Private helper method that removes the oldest element from the list based on the
fill direction. This method is called by Push() when the buffer is full to make
space for a new element.

### Operation
- fillFromLeft = TRUE: Oldest at end (high index), uses PopRight
- fillFromLeft = FALSE: Oldest at front (index 0), uses PopLeft

The removed element is discarded as we only care about making space.

### Return Value
- **TRUE**: Oldest element was successfully removed
- **FALSE**: Remove operation failed

### Side Effects
- Removes one element from the list
- May shift remaining elements (fillFromLeft = FALSE)
- Decrements element count by 1
- Increases available capacity by 1
*)
removeOldest := FALSE;
IF _reversed THEN
	// Fill from left: oldest element is at the end (highest index)
	removeOldest := anyBuffer.PopRight(dummyElement, TRUE);
ELSE
	// Fill from right: oldest element is at the front (index 0)
	removeOldest := anyBuffer.PopLeft(dummyElement, TRUE);
END_IF
END_METHOD

END_FUNCTION_BLOCK

// ---- Utilities/AnyBuffer/TypedBuffers/RingBuffer.TcPOU
// Provides a circular buffer (ring buffer) interface with automatic overwrite capability
FUNCTION_BLOCK RingBuffer IMPLEMENTS I_AnyBufferStrategy
VAR
	anyBuffer	  : I_AnyBuffer;
	isInitialized : BOOL := FALSE;
	_overwrite	  : BOOL := TRUE; // TRUE: overwrites oldest when full
END_VAR

(*
## Detailed Description

RingBuffer is an adapter that wraps an AnyBuffer instance to provide circular buffer
(also called ring buffer) semantics with automatic overwrite capability. When the buffer
is full and a new element is added, the oldest element is automatically removed to make
space, creating a continuous circular data flow.

### Alternative Names
This data structure is commonly known as:
- **Ring Buffer**: Emphasizes the circular/wrap-around nature
- **Circular Buffer**: Describes the logical circular structure
- **Cyclic Buffer**: Another term for the same concept

### Design Pattern
This implements the **Adapter Pattern**, which:
- Wraps the AnyBuffer interface with domain-specific circular buffer semantics
- Delegates all operations to the underlying AnyBuffer instance
- Provides automatic overwrite behavior when buffer reaches capacity
- Useful for streaming data, logging, and producer-consumer patterns

### Ring Buffer Semantics
- **Push(element)**: Adds element using circular indexing (FIFO enqueue)
  - When not full: Uses WriteAtIndex for direct write at tail position
  - When full: Overwrites oldest element using WriteAtIndex (no shifting!)
- **Pop(element)**: Removes oldest element using PeekAtIndex and circular head pointer (no shifting!)
- **Automatic overwrite**: When enabled and buffer is full, oldest data is overwritten in place
- **Circular indexing**: Uses head/tail pointers to track logical queue positions
- **Direct memory access**: Uses WriteAtIndex for O(1) writes without counter overhead
- Elements maintain FIFO order (first in, first out)

### Operation Mapping
```
Push() when not full  -> anyBuffer.WriteAtIndex(tail, ...)  // Direct write (O(1), no counter overhead)
Push() when full      -> anyBuffer.WriteAtIndex(tail, ...)  // Overwrite oldest (O(1), no shift!)
Pop()                 -> anyBuffer.PeekAtIndex(head, ...)   // Read oldest (O(1), no shift!)
Clear()               -> anyBuffer.Clear()                  // Clear all + reset indices
isEmpty               -> (elementCount = 0)                 // Check element count
isFull                -> (elementCount >= capacity)         // Check element count
```

### Usage Example
```iecst
VAR
    rawBuffer : ARRAY[0..2] OF DINT;  // Small buffer for demonstration
    buffer : AnyBuffer(pBuffer := rawBuffer,
                       bufferBoundLower := 0,
                       bufferBoundUpper := 2,
                       isBufferPersistent := FALSE);
    ring : RingBuffer(anyBuffer := buffer, overwrite := TRUE);
    value : DINT;
END_VAR

// Fill buffer
value := 100; ring.Push(value);  // Buffer: [100]
value := 200; ring.Push(value);  // Buffer: [100, 200]
value := 300; ring.Push(value);  // Buffer: [100, 200, 300] (full)

// Push to full buffer - oldest (100) is automatically removed
value := 400; ring.Push(value);  // Buffer: [200, 300, 400]
value := 500; ring.Push(value);  // Buffer: [300, 400, 500]

// Pop retrieves in FIFO order
ring.Pop(value);  // value = 300, Buffer: [400, 500]
```

### Circular Buffer Visualization
```
Initial state (capacity 5):
[ ][ ][ ][ ][ ]

After pushing 100, 200, 300:
[100][200][300][ ][ ]

After filling completely (100, 200, 300, 400, 500):
[100][200][300][400][500]  <- Full

After pushing 600 (overwrites 100):
[600][200][300][400][500]
     ^                ^
   oldest          newest

After pushing 700 (overwrites 200):
[600][700][300][400][500]
          ^             ^
       oldest       newest
```

### Advantages
- **No data loss when streaming**: Automatically maintains most recent data
- **Constant memory usage**: Buffer size never grows beyond capacity
- **Highly efficient**: Both Push and Pop are O(1) with circular indexing (no shifting!)
- **Simple interface**: Push/Pop semantics like FifoBuffer
- **Predictable behavior**: Always keeps newest data when overwrite is enabled
- **True circular buffer**: Implements proper ring buffer with head/tail pointers

### Use Cases
- **Logging buffers**: Keep most recent N log messages
- **Sensor data streams**: Store latest readings, discard old data
- **Audio/video buffers**: Maintain continuous data flow
- **Producer-consumer patterns**: Decouple data production and consumption rates
- **History tracking**: Keep fixed-size history of events or states

### Comparison with FifoBuffer
| Feature | FifoBuffer | RingBuffer |
|---------|-----------|------------|
| Behavior when full | Rejects new elements | Overwrites oldest |
| Push operation | Fails if full | Always succeeds |
| Data loss | Never (rejects push) | Yes (by design) |
| Use case | Queue with backpressure | Streaming data |
| Memory | Fixed size | Fixed size |

### Overwrite Behavior
- **overwrite = TRUE**: Push to full buffer removes oldest, adds newest (circular)
- **overwrite = FALSE**: Push to full buffer fails (same as FifoBuffer)

### Limitations
- No random access: Cannot peek at arbitrary indices (use AnyBuffer directly if needed)
- Overwrite is automatic: Cannot prevent data loss when buffer is full (by design)
- No notification: Caller is not informed when overwrite occurs

### Dependencies
- Requires I_AnyBuffer implementation (e.g., AnyBuffer)
- Uses Trace for error logging and verbose diagnostics
- Implements I_AnyBufferStrategy interface

### Performance Considerations
- **Push when not full**: O(1) - uses AppendRight
- **Push when full**: O(1) - uses ReplaceAtIndex with circular indexing (no shifting!)
- **Pop**: O(1) - uses PeekAtIndex with circular indexing (no shifting!)
- **Overall**: True O(1) constant-time operations for all Push and Pop operations
- Ideal for high-performance scenarios with frequent overwrites and streaming data

### Related Patterns
- **FifoBuffer**: FIFO queue without overwrite (rejects when full)
- **LifoBuffer**: Stack (Last-In-First-Out) semantics
- **PriorityBuffer**: Priority queue with ordered insertion
*)

METHOD PRIVATE AdvanceHead
// Advance tail pointer (circular)
anyBuffer.Metadata.headIndex := anyBuffer.Metadata.headIndex + 1;
IF anyBuffer.Metadata.headIndex > anyBuffer.Configuration.bufferBoundUpper THEN
	anyBuffer.Metadata.headIndex := anyBuffer.Configuration.bufferBoundLower;
END_IF
END_METHOD

METHOD PRIVATE AdvanceTail
// Advance tail pointer (circular)
anyBuffer.Metadata.tailIndex := anyBuffer.Metadata.tailIndex + 1;
IF anyBuffer.Metadata.tailIndex > anyBuffer.Configuration.bufferBoundUpper THEN
	anyBuffer.Metadata.tailIndex := anyBuffer.Configuration.bufferBoundLower;
END_IF
END_METHOD

// Removes all elements from the ring buffer and resets to empty state
METHOD Clear : BOOL

(*
## Detailed Description

Clears all elements from the underlying buffer, resetting it to an empty state.
After calling Clear, isEmpty will return TRUE and elementCount will be 0.

This operation delegates directly to the underlying anyBuffer.Clear() method.

### Return Value
- **TRUE**: Ring buffer was successfully cleared
- **FALSE**: Clear operation failed (e.g., anyBuffer is not initialized)

### Side Effects
- All elements are removed from the buffer
- Element count is reset to 0
- Buffer capacity is restored to maximum
- Logs verbose trace message on success
*)
Clear := FALSE;
IF anyBuffer <> 0 THEN
	Clear := anyBuffer.Clear();

	// Reset circular buffer indices
	anyBuffer.Metadata.headIndex	:= anyBuffer.Configuration.bufferBoundLower;
	anyBuffer.Metadata.tailIndex	:= anyBuffer.Configuration.bufferBoundLower;
	anyBuffer.Metadata.elementCount := 0;
END_IF

Trace.Verbose(__POUNAME(), 'executed');
END_METHOD

// Initializes the ring buffer by injecting the underlying buffer dependency
METHOD FB_Init : BOOL
VAR_INPUT
	bInitRetains : BOOL;		 // TRUE: the retain variables are initialized (reset warm / reset cold)
	bInCopyCode	 : BOOL;		 // TRUE: the instance will be copied to the copy code afterward (online change)
	anyBuffer	 : I_AnyBuffer;	 // The underlying buffer implementation to wrap
	overwrite	 : BOOL := TRUE; // TRUE: overwrites oldest element when full (circular behavior)
END_VAR

(*
## Detailed Description

Initializes the RingBuffer by injecting the underlying AnyBuffer dependency. This follows
the dependency injection pattern where the buffer implementation is provided during
construction rather than being created internally.

### Initialization Sequence
1. Validates that a valid anyBuffer reference is provided (non-zero pointer)
2. Stores the buffer reference for use by Push, Pop, and other operations
3. Stores the overwriteEnabled flag to control circular buffer behavior
4. Sets isInitialized flag to TRUE to enable operations

### Parameters
- **anyBuffer**: Reference to an I_AnyBuffer implementation (e.g., AnyBuffer instance)
  - Must be a valid, initialized buffer
  - This RingBuffer will delegate all operations to this buffer
- **overwriteEnabled**: Controls behavior when buffer is full
  - **TRUE** (default): Push to full buffer removes oldest, adds newest (circular behavior)
  - **FALSE**: Push to full buffer fails and logs error (same as FifoBuffer)

### Return Value
Returns BOOL but value is not evaluated by the runtime. Always call with valid anyBuffer.

### Usage Example
```iecst
VAR
    rawBuffer : ARRAY[0..9] OF DINT;
    buffer : AnyBuffer(pBuffer := rawBuffer,
                       bufferBoundLower := 0,
                       bufferBoundUpper := 9,
                       isBufferPersistent := FALSE);
    ring : RingBuffer(anyBuffer := buffer,
                      overwriteEnabled := TRUE);  // Enable circular overwrite
END_VAR
```

### Important Notes
- Must provide a valid anyBuffer reference, otherwise Push/Pop will fail
- The underlying buffer must already be initialized before passing to FB_Init
- Setting overwriteEnabled to FALSE makes RingBuffer behave like FifoBuffer
*)
IF anyBuffer <> 0 THEN
	THIS^.anyBuffer	 := anyBuffer;
	THIS^._overwrite := _overwrite;
	isInitialized	 := TRUE;
END_IF
END_METHOD

// Returns TRUE if the ring buffer contains no elements
PROPERTY isEmpty : BOOL

(*
## Detailed Description

Returns TRUE if the ring buffer is empty (contains no elements), FALSE otherwise.
This property delegates directly to the underlying anyBuffer.isEmpty property.

Use this property to check if Pop operation would succeed before attempting to
remove an element.

### Return Value
- **TRUE**: Ring buffer is empty (elementCount = 0)
- **FALSE**: Ring buffer contains one or more elements

### Usage Example
```iecst
IF NOT ring.isEmpty THEN
    ring.Pop(value);  // Safe to pop
END_IF
```
*)
GET
isEmpty := (anyBuffer.Metadata.elementCount = 0);
END_GET
END_PROPERTY

// Returns TRUE if the ring buffer is at maximum capacity
PROPERTY isFull : BOOL

(*
## Detailed Description

Returns TRUE if the ring buffer is full (at maximum capacity), FALSE otherwise.
This property delegates directly to the underlying anyBuffer.isFull property.

Note: When overwriteEnabled is TRUE, Push will still succeed even when isFull is TRUE
by automatically removing the oldest element. When overwriteEnabled is FALSE, Push
will fail when isFull is TRUE.

### Return Value
- **TRUE**: Ring buffer is full (elementCount = capacity)
- **FALSE**: Ring buffer has space for more elements

### Usage Example
```iecst
IF ring.isFull THEN
    // With overwriteEnabled=TRUE, Push will overwrite oldest
    // With overwriteEnabled=FALSE, Push will fail
    value := 100;
    success := ring.Push(value);
END_IF
```
*)
GET
isFull := (anyBuffer.Metadata.elementCount >= anyBuffer.Configuration.capacity);
END_GET
END_PROPERTY

// Removes and retrieves the oldest element from the ring buffer (FIFO dequeue)
{attribute 'hasanytype'}
METHOD Pop : BOOL
VAR_INPUT
	element : ANY; // Variable to receive the popped element
END_VAR

(*
## Detailed Description

Removes and retrieves the oldest element from the ring buffer following FIFO (First-In-First-Out)
semantics. The element that was pushed first (or oldest remaining after overwrites) is removed
and copied to the provided element parameter.

This operation uses anyBuffer.PeekAtIndex() to read the element at the head position, then
advances the head pointer circularly. No element shifting occurs, making this an O(1) operation.

### Operation Sequence
1. Validates that the buffer has been initialized
2. Validates that element size matches the buffer's configured element size
3. Checks that the ring buffer is not empty
4. Reads element at head position using PeekAtIndex (no removal, no shifting!)
5. Copies the element value to the output parameter
6. Advances head pointer circularly: headIndex = (headIndex + 1) MOD capacity
7. Decrements element count
8. Logs verbose trace on success or error trace on failure

### FIFO Behavior Example
```iecst
value := 100; ring.Push(value);  // Buffer: [100]
value := 200; ring.Push(value);  // Buffer: [100, 200]
value := 300; ring.Push(value);  // Buffer: [100, 200, 300]

ring.Pop(value);  // Returns 100 (oldest), Buffer: [200, 300]
ring.Pop(value);  // Returns 200 (next oldest), Buffer: [300]
ring.Pop(value);  // Returns 300 (last), Buffer: []
```

### Return Value
- **TRUE**: Element was successfully popped and copied to element parameter
- **FALSE**: Pop operation failed (see error conditions)

### Error Conditions
- Returns FALSE and logs error if buffer was not initialized
- Returns FALSE and logs error if element size doesn't match buffer element size
- Returns FALSE and logs error if ring buffer is empty (no elements to pop)
- Returns FALSE and logs error if underlying PopLeft operation fails

### Parameters
- **element**: Must be a writable variable (not a literal) of the correct size
  - Must match the buffer's configured element size
  - Will receive the popped element value on success

### Side Effects
- Logically removes one element from the ring buffer (advances head pointer)
- No physical shifting of elements occurs
- Decrements element count by 1
- Advances head pointer circularly
- Logs verbose trace message on success
- Logs error trace message on failure

### Performance Considerations
- **Time complexity**: O(1) - constant time operation
- No element shifting required due to circular indexing
- Optimal performance for ring buffer operations
*)
Pop := FALSE;
IF NOT isInitialized THEN
	Trace.Error(__POUNAME(), 'Buffer was not initialized yet, execute method .init() at least once');
	RETURN;
END_IF

// valid sized element pushed?
IF element.diSize <> anyBuffer.Configuration.elementSize THEN
	Trace.Error(__POUNAME(), 'Passed element to pop to is of improper size');
	RETURN;
END_IF

// retrieve element at the head position if there is any left in the buffer
IF NOT isEmpty THEN
	// Read and clear element at head position (no shifting!)
	Pop := anyBuffer.PeekAtIndex(anyBuffer.Metadata.headIndex, element);
	IF Pop THEN
		anyBuffer.DeleteAtIndex(anyBuffer.Metadata.headIndex);

		// Delete index does not change counters, do it manually
		anyBuffer.Metadata.capacity		:= anyBuffer.Metadata.capacity + 1;
		anyBuffer.Metadata.elementCount := anyBuffer.Metadata.elementCount - 1;

		// Advance head circular
		AdvanceHead();
	END_IF
ELSE
	Trace.Error(__POUNAME(), 'Attempt to pop from empty buffer');
END_IF

// Pop was ok, trace message
IF Pop THEN
	Trace.Verbose(__POUNAME(), 'executed');
ELSE
	Trace.Error(__POUNAME(), 'FAILED');
END_IF
END_METHOD

// Adds a new element to the ring buffer with optional automatic overwrite
{attribute 'hasanytype'}
METHOD Push : BOOL
VAR_INPUT
	element : ANY; // Element to add to the ring buffer
END_VAR

VAR
	dummyElement : AnyType; // For discarding oldest element
END_VAR

(*
## Detailed Description

Adds a new element to the ring buffer. Behavior depends on the overwriteEnabled setting:

**When overwriteEnabled = TRUE (circular buffer mode)**:
- If buffer is not full: Adds element using WriteAtIndex (direct write at tail position)
- If buffer is full: Overwrites oldest element at tail position using WriteAtIndex (no shifting!)
- Push always succeeds (except for validation errors)
- Oldest data is automatically overwritten in place when buffer is full
- Both head and tail pointers advance circularly
- No buffer counter updates (managed by RingBuffer)

**When overwriteEnabled = FALSE (bounded queue mode)**:
- If buffer is not full: Adds element using WriteAtIndex
- If buffer is full: Operation fails and logs error
- Behaves like a bounded queue (rejects new elements when full)

### Operation Sequence (overwriteEnabled = TRUE)
1. Validates that the buffer has been initialized
2. Validates that element size matches the buffer's configured element size
3. If buffer not full: Uses WriteAtIndex and advances tail pointer, increments elementCount
4. If buffer is full: Overwrites at tail position using WriteAtIndex, advances both head and tail circularly
5. No element shifting occurs, no AnyBuffer counter changes
6. Logs verbose trace on success or error trace on failure

### Operation Sequence (overwriteEnabled = FALSE)
1. Validates that the buffer has been initialized
2. Validates that element size matches the buffer's configured element size
3. Checks that buffer is not full
4. Adds new element at tail position using WriteAtIndex
5. Logs verbose trace on success or error trace on failure

### Circular Buffer Example (overwriteEnabled = TRUE)
```iecst
// Buffer capacity = 3
value := 100; ring.Push(value);  // Buffer: [100]
value := 200; ring.Push(value);  // Buffer: [100, 200]
value := 300; ring.Push(value);  // Buffer: [100, 200, 300] (full)

// Push to full buffer - oldest (100) is removed automatically
value := 400; ring.Push(value);  // Buffer: [200, 300, 400]
value := 500; ring.Push(value);  // Buffer: [300, 400, 500]

// Latest 3 elements are always retained
```

### Bounded Queue Example (overwriteEnabled = FALSE)
```iecst
// Buffer capacity = 3
value := 100; ring.Push(value);  // Buffer: [100], returns TRUE
value := 200; ring.Push(value);  // Buffer: [100, 200], returns TRUE
value := 300; ring.Push(value);  // Buffer: [100, 200, 300], returns TRUE

// Push to full buffer fails
value := 400;
success := ring.Push(value);     // Returns FALSE, logs error, buffer unchanged
```

### Return Value
- **TRUE**: Element was successfully pushed to the ring buffer
- **FALSE**: Push operation failed (see error conditions)

### Error Conditions (both modes)
- Returns FALSE and logs error if buffer was not initialized
- Returns FALSE and logs error if element size doesn't match buffer element size
- Returns FALSE and logs error if underlying WriteAtIndex operation fails

### Error Conditions (overwriteEnabled = FALSE only)
- Returns FALSE and logs error if ring buffer is full (no available capacity)

### Parameters
- **element**: Must be a writable variable (not a literal) of the correct size
  - Must match the buffer's configured element size
  - Value will be copied into the ring buffer

### Side Effects (when not full)
- Adds one element to the ring buffer using WriteAtIndex
- Increments elementCount by 1 (managed by RingBuffer, not AnyBuffer)
- Advances tail pointer circularly
- Logs verbose trace message on success
- Logs error trace message on failure

### Side Effects (when full and overwriteEnabled = TRUE)
- Overwrites element at tail position using WriteAtIndex (no shifting!)
- Advances both head pointer and tail pointer circularly
- Element count remains at maximum capacity
- No physical element movement occurs
- No AnyBuffer counter modifications
- Logs verbose trace message on success

### Performance Considerations
- **When not full**: O(1) - uses WriteAtIndex (raw write, no counter overhead)
- **When full**: O(1) - uses WriteAtIndex with circular indexing (no shifting!)
- **Overall**: True O(1) constant-time operation for all scenarios
- **Optimal efficiency**: WriteAtIndex bypasses AnyBuffer counter management
- Ideal for high-frequency streaming and real-time data processing
*)
Push := FALSE;
IF NOT isInitialized THEN
	Trace.Error(__POUNAME(), 'Buffer was not initialized yet, execute method .init() at least once');
	RETURN;
END_IF

// valid sized element pushed?
IF element.diSize <> anyBuffer.Configuration.elementSize THEN
	Trace.Error(__POUNAME(), 'Pushed element is of improper size');
	RETURN;
END_IF

// Handle push based on buffer state
IF anyBuffer.Metadata.elementCount < anyBuffer.Configuration.capacity THEN
	// Buffer not yet full - use WriteAtIndex for direct write without counter changes
	Push := anyBuffer.ReplaceAtIndex(anyBuffer.Metadata.tailIndex, element);
	IF Push THEN
		// Advance tail circular
		AdvanceTail();

		// Replace index does not change counters, do it manually
		anyBuffer.Metadata.elementCount := anyBuffer.Metadata.elementCount + 1;
		anyBuffer.Metadata.capacity		:= anyBuffer.Metadata.capacity - 1;
	END_IF
ELSIF _overwrite THEN
	// Buffer is full and overwrite enabled - use WriteAtIndex for circular overwrite (no shifting!)
	Push := anyBuffer.ReplaceAtIndex(anyBuffer.Metadata.tailIndex, element);
	IF Push THEN
		// Advance tail circular
		AdvanceTail();

		// Advance head circular
		AdvanceHead();

		// elementCount stays at capacity
	END_IF
ELSE
	// Overwrite disabled - reject push when full (bounded queue behavior)
	Trace.Error(__POUNAME(), 'Attempt to push to full buffer with overwrite disabled');
	RETURN;
END_IF

// Push was ok, trace message
IF Push THEN
	Trace.Verbose(__POUNAME(), 'executed');
ELSE
	Trace.Error(__POUNAME(), 'FAILED');
END_IF
END_METHOD

END_FUNCTION_BLOCK

// ---- Utilities/File/File_HMI.TcPOU
FUNCTION_BLOCK File_HMI EXTENDS HmiFunction
VAR
	File : I_FileHandler;
	{ attribute 'TcHmiSymbol.AddSymbol' }
	{ attribute 'TcHmiSymbol.AddSymbol.UserGroups' := '__SystemAdministrators,Admin' }
	File_HMI : ST_File_HMI;
END_VAR

PROPERTY ControlObject : I_Base
SET
__QueryInterface(ControlObject,File);
END_SET
END_PROPERTY

METHOD CyclicLogic
VAR_INST
	SaveRT		 : R_TRIG;
	LoadRT		 : R_TRIG;
	ReloadActive : BOOL;
END_VAR
IF File = 0 THEN
	RETURN;
END_IF

File_HMI.Name		:= File.Name;
File_HMI.HmiEnabled := Enabled;
// HMI Commands
IF Enabled THEN
	SaveRT(CLK := File_HMI.Save.Active);
	IF SaveRT.Q THEN
		IF File_HMI.Save.Permissive.OK THEN
			File.UpdateSymbol();
		END_IF
	END_IF

	IF ReloadActive AND NOT File.Busy AND NOT File.Error THEN
		File.ReadSymbol();
		ReloadActive := FALSE;
	END_IF

	LoadRT(CLK := File_HMI.Load.Active);
	IF LoadRT.Q THEN
		IF File_HMI.Load.Permissive.OK THEN
			File.LoadFile();
			ReloadActive := TRUE;
		END_IF
	END_IF

	IF File_HMI.NewPath THEN
		File.Path		 := File_HMI.Path;
		File_HMI.NewPath := FALSE;
	END_IF
END_IF
END_METHOD

(*FB_Init is always available implicitly and it is used primarily for initialization.
The return value is not evaluated. For a specific influence, you can also declare the
methods explicitly and provide additional code there with the standard initialization
code. You can evaluate the return value.*)
METHOD FB_Init : BOOL
VAR_INPUT
	(* TRUE: the retain variables are initialized (reset warm / reset cold)*)
	bInitRetains : BOOL;

	(* TRUE: the instance will be copied to the copy code afterward (online change)   *)
	bInCopyCode : BOOL;
	Name		: T_MaxString;
	File		: I_FileHandler;
END_VAR
THIS^.File	:= File;
ControlType := 'File';
LinkObject	:= 'File_HMI';
END_METHOD

PROPERTY LoadPermissive : I_Permissive
GET
LoadPermissive := File_HMI.Load.Permissive;
END_GET
END_PROPERTY

PROPERTY SavePermissive : I_Permissive
GET
SavePermissive := File_HMI.Save.Permissive;
END_GET
END_PROPERTY

END_FUNCTION_BLOCK

// ---- Utilities/File/JsonFile.TcPOU
FUNCTION_BLOCK JsonFile
VAR_GENERIC CONSTANT
	FileSize : UDINT := 10000;
END_VAR
EXTENDS CyclicComponent IMPLEMENTS I_FileHandler
VAR
	{attribute 'hide'}
	_Error : BOOL;
	{attribute 'hide'}
	_ErrorId : UDINT;

	//
	_Path	   : STRING;
	TonTimeout : TON;
	_Timeout   : TIME := T#1S;
	SeqLoad	   : UDINT;
	SeqSave	   : UDINT;

	// Folder Management
	CreateDir	 : FB_CreateDir;
	StringHelper : StringHelper;

	// Symbol
	JsonReadWriteDataType : FB_JsonReadWriteDatatype;
	ValueJson			  : STRING(FileSize);
	hr					  : HRESULT;
	_Datatype			  : T_MaxString;
	_SymbolName			  : T_MaxString;
	_nData				  : UDINT;
	_pData				  : PVOID;

	// Json Management 
	FileRead			  : BOOL;
	FileSave			  : BOOL;
	FileLoadOK			  : BOOL;
	FileSaveOK			  : BOOL;
	JsonFileMachineConfig : FB_JsonDomParser;
	JsonDoc				  : SJsonValue;
	JsonProp			  : SJsonValue;
END_VAR

{attribute 'monitoring' := 'call'}
PROPERTY Busy : BOOL
GET
Busy := SeqSave <> 0 OR SeqLoad <> 0;
END_GET
END_PROPERTY

METHOD ClearDocument
VAR_INPUT
END_VAR
JsonDoc := JsonFileMachineConfig.NewDocument();
END_METHOD

METHOD CyclicLogic
IF _Path <> '' THEN
	FileLoadOK := JsonFileMachineConfig.LoadDocumentFromFile(sFile := _Path, bExec := FileRead);
	FileSaveOK := JsonFileMachineConfig.SaveDocumentToFile(sFile := _Path, bExec := FileSave);
END_IF

TonTimeout(IN := Busy, PT := _Timeout);
IF TonTimeout.Q THEN
	_Error := TRUE;
END_IF

SaveFileSequence();
LoadFileSequence();
END_METHOD

PROPERTY Datatype : T_MaxString
SET
_Datatype := Datatype;
END_SET
END_PROPERTY

{attribute 'monitoring' := 'call'}
PROPERTY Error : BOOL
GET
Error := _Error;
END_GET
END_PROPERTY

{attribute 'monitoring' := 'call'}
PROPERTY ErrorId : UDINT
GET
ErrorID := _ErrorID;
END_GET
END_PROPERTY

METHOD LoadFile
IF _Path = '' THEN
	_Error := TRUE;
	Trace.LogMessage(Name, 'File Path not set!');
	RETURN;
END_IF

IF Busy THEN
	RETURN;
END_IF

FileRead := TRUE;
SeqLoad	 := 10;
END_METHOD

METHOD PRIVATE LoadFileSequence
VAR_INST
	dirPath	 : T_MaxString;
	tryAgain : BOOL;
END_VAR

VAR
	msg : STRING;
END_VAR
CASE SeqLoad OF
	0:										// Attempt to Load File -> Command started in LoadFile()
	10:										// Load File Done
		IF NOT FileRead AND FileLoadOK THEN // File Found
			JsonDoc := JsonFileMachineConfig.GetDocumentRoot();
			SeqLoad := 0;
		END_IF

		IF (NOT FileRead AND NOT FileLoadOK) OR TonTimeout.Q THEN // File not Found
			tryAgain := FALSE;
			FileRead := FALSE;
			SeqLoad	 := 20;
		END_IF

	20:								  (*File Not Found - Create Directory if not exists*) ;
		CreateDir(bExecute := FALSE); //Prepare for rising edge in next step
		IF NOT tryAgain THEN
			dirPath := StringHelper.GetPath(_Path);
		ELSE
			dirPath := StringHelper.GetPath(dirPath);
		END_IF

		SeqLoad := 30;

	30:
		CreateDir(sNetId	:= '',
				  sPathName := dirPath,
				  ePath		:= PATH_GENERIC,
				  bExecute	:= TRUE);

		IF NOT CreateDir.bBusy THEN
			IF NOT CreateDir.bError THEN
				IF NOT tryAgain THEN
					SeqLoad := 40;
				ELSE
					tryAgain := FALSE;
					SeqLoad	 := 20;
				END_IF
			ELSE
				IF (CreateDir.nErrId = 1827) OR (CreateDir.nErrId = 1807) THEN
					//0x723 Folder is already existing or invalid sPathName or ePath parameter.
					msg := CONCAT(_Path, ' File not found, but folder is existing. File will be created');
					Trace.LogMessage(Name, msg);
					SeqLoad := 40;
				ELSIF CreateDir.nErrId = 1804 THEN
					//0x70C Folder not found.
					msg := CONCAT('Folder is not found: ', dirPath);
					msg := CONCAT(msg, ' Reducing Path and trying again.');
					Trace.LogMessage(Name, msg);
					tryagain := TRUE;

					// SeqLoad	 := 20; TwinCat Bug - Ticket BTS-168764 Germany
					SeqLoad := 40;
				ELSE
					msg := CONCAT('Create Directory Error: ', UDINT_TO_STRING(CreateDir.nErrId));
					Trace.LogMessage(Name, msg);
					SeqLoad := 999;
				END_IF
			END_IF
		END_IF

	40: // File not found -> Create file
		JsonDoc	 := JsonFileMachineConfig.NewDocument();
		FileSave := TRUE;
		SeqLoad	 := 50;

	50: // New Document Saved
		IF NOT FileSave AND FileSaveOk THEN
			_Error	:= FALSE;
			SeqLoad := 0;
		END_IF
END_CASE
END_METHOD

PROPERTY nData : UDINT
SET
_nData := nData;
END_SET
END_PROPERTY

PROPERTY PUBLIC Path : T_MaxString
GET
Path := _Path;
END_GET
SET
//Prevent the path from have a space at the end
_Path := Path;
WHILE RIGHT(_Path, 1) = ' ' DO
	_Path := DELETE(_Path, 1, LEN(_Path));
END_WHILE
END_SET
END_PROPERTY

PROPERTY pData : PVOID
SET
_pData := pData;
END_SET
END_PROPERTY

METHOD ReadSymbol
IF JsonDoc = 0 THEN
	Trace.LogMessage(Name, 'Document File not loaded!');
	RETURN;
END_IF

IF _Datatype = '' THEN
	Trace.LogMessage(Name, 'No Datatype specified!');
	RETURN;
END_IF

IF _nData = 0 THEN
	Trace.LogMessage(Name, 'No nData specified!');
	RETURN;
END_IF

IF _pData = 0 THEN
	Trace.LogMessage(Name, 'No pData specified!');
	RETURN;
END_IF

IF _SymbolName = '' THEN
	Trace.LogMessage(Name, 'No PropertyName specified!');
	RETURN;
END_IF

IF Busy THEN
	RETURN;
END_IF

JsonProp := JsonFileMachineConfig.FindMemberPath(JsonDoc, _SymbolName);
JsonFileMachineConfig.CopyJson(v := JsonProp, pDoc := ValueJson, nDoc := SIZEOF(ValueJson));
IF JsonProp <> 0 THEN
	JsonReadWriteDataType.SetSymbolFromJson(sJson		:= ValueJson,
											sDataType	:= _Datatype,
											nData		:= _nData,
											pData		:= _pData,
											hrErrorCode => hr);
ELSE
	THIS^.UpdateSymbol();
END_IF
END_METHOD

METHOD Reset
_Error		  := FALSE;
_ErrorId	  := 0;
SeqSave		  := 0;
SeqLoad		  := 0;
TonTimeout.IN := FALSE;
END_METHOD

METHOD SaveFile
IF _Path = '' THEN
	_Error := TRUE;
	Trace.LogMessage(Name, 'File Path not set!');
	RETURN;
END_IF

IF Busy THEN
	RETURN;
END_IF

FileSave := TRUE;
SeqSave	 := 10;
END_METHOD

METHOD PRIVATE SaveFileSequence
CASE SeqSave OF
	0:	// Attempt to save File -> Command started in UpdateXYZ()
	10: // New Document Saved
		IF NOT FileSave AND FileSaveOk THEN
			SeqSave := 0;
		END_IF
END_CASE
END_METHOD

PROPERTY SymbolName : T_MaxString
SET
_SymbolName := SymbolName;
END_SET
END_PROPERTY

PROPERTY Timeout : TIME
SET
_Timeout := Timeout;
END_SET
END_PROPERTY

METHOD UpdateSymbol
IF JsonDoc = 0 THEN
	Trace.LogMessage(Name, 'Document File not loaded!');
	RETURN;
END_IF

IF _Datatype = '' THEN
	Trace.LogMessage(Name, 'No Datatype specified!');
	RETURN;
END_IF

IF _nData = 0 THEN
	Trace.LogMessage(Name, 'No nData specified!');
	RETURN;
END_IF

IF _pData = 0 THEN
	Trace.LogMessage(Name, 'No pData specified!');
	RETURN;
END_IF

IF _SymbolName = '' THEN
	Trace.LogMessage(Name, 'No PropertyName specified!');
	RETURN;
END_IF

IF Busy THEN
	RETURN;
END_IF

// Create Json
JsonReadWriteDataType.CopyJsonStringFromSymbol(sDatatype   := _Datatype,
											   nData	   := _nData,
											   pData	   := _pData,
											   pDoc		   := ValueJson,
											   nDoc		   := SIZEOF(ValueJson),
											   hrErrorCode => hr);

// Attempt to find Member
jsonProp := JsonFileMachineConfig.FindMemberPath(JsonDoc, _SymbolName);
IF JsonProp <> 0 THEN
	JsonFileMachineConfig.SetJson(JsonProp, ValueJson);
ELSE
	JsonFileMachineConfig.AddJsonMember(JsonDoc, _SymbolName, ValueJson);
END_IF

// Save the update to file
FileSave := TRUE;
SeqSave	 := 10;
JsonProp := 0;
END_METHOD

END_FUNCTION_BLOCK

// ---- Utilities/File/StringHelper.TcPOU
{attribute 'no_explicit_call' := 'This FB is a CLASS and must be accessed using methods or properties'}
FUNCTION_BLOCK StringHelper

METHOD PROTECTED GetExtensionOrVarName : T_MaxString
VAR_INPUT
	input : T_MaxString;
END_VAR

VAR
	i		 : INT;
	charArry : ARRAY[0..255] OF STRING(1);
END_VAR
IF NOT ValidInput(input) THEN
	RETURN;
END_IF

charArry := StringToCharArray(input);
//Get Location of final delimiter '.'
FOR i := LEN(input) - 1 TO 0 BY -1 DO //Start at the end and find the last delimiter
	IF charArry[i] = '.' THEN
		GetExtensionOrVarName := RIGHT(input, LEN(input) - 1 - i);
		EXIT;
	END_IF
END_FOR
END_METHOD

METHOD PROTECTED GetFileNameFromPath : T_MaxString
VAR_INPUT
	input : T_MaxString;
END_VAR

VAR
	i			  : INT;
	searchResults : ARRAY[0..99] OF INT;
	tempPath	  : T_MaxString;
END_VAR
IF NOT ValidInput(input) THEN
	RETURN;
END_IF

tempPath := input; //Copy to temp variable for modification
FOR i := 0 TO LEN(input) - 1 DO
	searchResults[i] := FIND(tempPath, '\');
	IF searchResults[i] > 0 THEN
		tempPath := RIGHT(tempPath, LEN(tempPath) - searchResults[i]); //Remove begining up to and including the first delimiter
	ELSE
		EXIT; //No more delimiters remaining
	END_IF
END_FOR

GetFileNameFromPath := tempPath;
END_METHOD

METHOD PROTECTED GetFilePath : T_MaxString
VAR_INPUT
	input : T_MaxString;
END_VAR

VAR
	tempPath	  : T_MaxString;
	i			  : INT;
	searchResults : ARRAY[0..99] OF INT;
	location	  : INT;
END_VAR
IF NOT ValidInput(input) THEN
	RETURN;
END_IF

tempPath := input;								 //Copy to temp variable for modification
tempPath := LEFT(tempPath, (LEN(tempPath) - 1)); //Remove Last Character, on first pass this has no effect, but on subsequents passes this will remove the ending \

//Reduce String by removing each delimiter and counting number of characters removed to find last '\'
FOR i := 0 TO LEN(input) - 1 DO
	searchResults[i] := FIND(tempPath, '\');
	IF searchResults[i] > 0 THEN
		tempPath := RIGHT(tempPath, LEN(tempPath) - searchResults[i]); //Remove begining up to and including the first delimiter
	ELSE
		EXIT; //No more delimiters remaining
	END_IF
END_FOR

//Sum length of string to last delimiter
FOR i := 0 TO LEN(input) - 1 DO
	IF searchResults[i] > 0 THEN
		location := location + searchResults[i]; //Location of last delimiter
	ELSE
		EXIT;
	END_IF
END_FOR

GetFilePath := LEFT(input, location);
END_METHOD

METHOD GetName : T_MaxString
VAR_INPUT
	FullPath : T_MaxString;
END_VAR
IF NOT ValidInput(FullPath) THEN
	RETURN;
END_IF

//Find the First \ or . to determine if this is a File Path or Symbol Path
IF FIND(FullPath, '\') > 0 THEN
	GetName := GetFileNameFromPath(FullPath);
ELSE //symbolPath
	GetName := GetExtensionOrVarName(FullPath);
END_IF
END_METHOD

METHOD GetPath : T_MaxString
VAR_INPUT
	FullPath : T_MaxString;
END_VAR

VAR
	tempPath : T_MaxString;
END_VAR
IF NOT ValidInput(FullPath) THEN
	RETURN;
END_IF

//Find the First \ or . to determine if this is a File Path or Symbol Path
IF FIND(FullPath, '\') > 0 THEN
	GetPath := GetFilePath(FullPath);
ELSE //symbolPath
	GetPath := GetSymbolPath(FullPath);
END_IF
END_METHOD

METHOD PROTECTED GetSymbolPath : T_MaxString
VAR_INPUT
	input : T_MaxString;
END_VAR

VAR
	i		 : INT;
	charArry : ARRAY[0..255] OF STRING(1);
	tempPath : T_MaxString;
END_VAR
IF NOT ValidInput(input) THEN
	RETURN;
END_IF

charArry := StringToCharArray(input);
tempPath := input;					  //Copy to temp variable for modification
FOR i := LEN(input) - 1 TO 0 BY -1 DO //Start at the end and find the last delimiter
	IF charArry[i] = '.' THEN
		tempPath := LEFT(tempPath, i);
		EXIT;
	END_IF
END_FOR

GetSymbolPath := tempPath;
END_METHOD

METHOD PROTECTED RemoveFirstChar : T_MaxString
VAR_INPUT
	input : T_MaxString;
END_VAR
RemoveFirstChar := DELETE(input, 1, 1);
END_METHOD

METHOD PROTECTED RemoveLastChar : T_MaxString
VAR_INPUT
	input : T_MaxString;
END_VAR
RemoveLastChar := DELETE(input, 1, len(input));
END_METHOD

METHOD PROTECTED StringToCharArray : ARRAY[0..255] OF STRING(1)
VAR_INPUT
	input : T_MaxString;
END_VAR

VAR
	i		 : INT;
	end		 : INT;
	tempPath : T_MaxString;
END_VAR
IF NOT ValidInput(input) THEN
	RETURN;
END_IF

tempPath := input;
//Convert String to CharArray
FOR i := 0 TO LEN(input) - 1 DO
	StringToCharArray[i] := Left(tempPath, 1); //Return the first/next character
	tempPath			 := RemoveFirstChar(tempPath);
END_FOR
END_METHOD

METHOD PROTECTED ValidInput : BOOL
VAR_INPUT
	input : T_MaxString;
END_VAR
IF LEN(input) > 0 THEN
	ValidInput := TRUE;
ELSE
	ValidInput := FALSE;
END_IF
END_METHOD

END_FUNCTION_BLOCK

// ---- Utilities/Flash/SyncedSquareWaves.TcPOU
FUNCTION_BLOCK SyncedSquareWaves EXTENDS CyclicComponent IMPLEMENTS I_Initializable
VAR
	_Initialized  : BOOL;
	PLC_CycleTime : UDINT;
	CycleTime_ms  : LREAL;

	//
	{attribute 'hide'}
	_Wave_500Hz : BOOL;
	{attribute 'hide'}
	_Wave_100Hz : BOOL;
	{attribute 'hide'}
	_Wave_50Hz : BOOL;
	{attribute 'hide'}
	_Wave_5Hz : BOOL;
	{attribute 'hide'}
	_Wave_2Hz : BOOL;
	{attribute 'hide'}
	_Wave_1Hz : BOOL;
	{attribute 'hide'}
	_Wave_0_5Hz : BOOL;
END_VAR

//! @summary This method serves as the entry point for all underlying FB logic
METHOD PUBLIC CyclicLogic
VAR
	Counter		   : LREAL;
	CountsRequired : LREAL;
	CycleCount	   : UDINT;
END_VAR
IF NOT _Initialized THEN
	Initialize();
	RETURN;
END_IF

CycleCount := TwinCAT_SystemInfoVarList._TaskInfo[GETCURTASKINDEXEX()].CycleCount;
IF (CycleTime_ms <= 1) AND (FRAC(1 / CycleTime_ms) = 0) THEN
	CountsRequired := 1 / CycleTime_ms;
	Counter		   := LMOD(CycleCount, CountsRequired);
	IF (Counter + 1) = CountsRequired THEN
		_Wave_500Hz := NOT _Wave_500Hz;
	END_IF
END_IF

IF (CycleTime_ms <= 5) AND (FRAC(5 / CycleTime_ms) = 0) THEN
	CountsRequired := 5 / CycleTime_ms;
	Counter		   := LMOD(CycleCount, CountsRequired);
	IF (Counter + 1) = CountsRequired THEN
		_Wave_100Hz := NOT _Wave_100Hz;
	END_IF
END_IF

IF (CycleTime_ms <= 10) AND (FRAC(10 / CycleTime_ms) = 0) THEN
	CountsRequired := 10 / CycleTime_ms;
	Counter		   := LMOD(CycleCount, CountsRequired);
	IF (Counter + 1) = CountsRequired THEN
		_Wave_50Hz := NOT _Wave_50Hz;
	END_IF
END_IF

IF (CycleTime_ms <= 100) AND (FRAC(100 / CycleTime_ms) = 0) THEN
	CountsRequired := 100 / CycleTime_ms;
	Counter		   := LMOD(CycleCount, CountsRequired);
	IF (Counter + 1) = CountsRequired THEN
		_Wave_5Hz := NOT _Wave_5Hz;
	END_IF
END_IF

IF (CycleTime_ms <= 250) AND (FRAC(250 / CycleTime_ms) = 0) THEN
	CountsRequired := 250 / CycleTime_ms;
	Counter		   := LMOD(CycleCount, CountsRequired);
	IF (Counter + 1) = CountsRequired THEN
		_Wave_2Hz := NOT _Wave_2Hz;
	END_IF
END_IF

IF (CycleTime_ms <= 500) AND (FRAC(500 / CycleTime_ms) = 0) THEN
	CountsRequired := 500 / CycleTime_ms;
	Counter		   := LMOD(CycleCount, CountsRequired);
	IF (Counter + 1) = CountsRequired THEN
		_Wave_1Hz := NOT _Wave_1Hz;
	END_IF
END_IF

IF (CycleTime_ms <= 1000) AND (FRAC(1000 / CycleTime_ms) = 0) THEN
	CountsRequired := 1000 / CycleTime_ms;
	Counter		   := LMOD(CycleCount, CountsRequired);
	IF (Counter + 1) = CountsRequired THEN
		_Wave_0_5Hz := NOT _Wave_0_5Hz;
	END_IF
END_IF
END_METHOD

METHOD Initialize
//PLC Scan Info
PLC_CycleTime := TwinCAT_SystemInfoVarList._TaskInfo[GETCURTASKINDEXEX()].CycleTime;
CycleTime_ms  := TO_LREAL(PLC_CycleTime) / 10000.0;

//
_Wave_500Hz	 := TRUE;
_Wave_100Hz	 := TRUE;
_Wave_50Hz	 := TRUE;
_Wave_5Hz	 := TRUE;
_Wave_2Hz	 := TRUE;
_Wave_1Hz	 := TRUE;
_Wave_0_5Hz	 := TRUE;
_Initialized := TRUE;
END_METHOD

{attribute 'monitoring' := 'call'}
PROPERTY Initialized : BOOL
GET
Initialized := _Initialized;
END_GET
SET
_Initialized := Initialized;
END_SET
END_PROPERTY

{attribute 'monitoring' := 'call'}
PROPERTY Wave_0_5Hz : BOOL
GET
Wave_0_5Hz := _Wave_0_5Hz;
END_GET
END_PROPERTY

{attribute 'monitoring' := 'call'}
PROPERTY Wave_100Hz : BOOL
GET
Wave_100Hz := _Wave_100Hz;
END_GET
END_PROPERTY

{attribute 'monitoring' := 'call'}
PROPERTY Wave_1Hz : BOOL
GET
Wave_1Hz := _Wave_1Hz;
END_GET
END_PROPERTY

{attribute 'monitoring' := 'call'}
PROPERTY Wave_2Hz : BOOL
GET
Wave_2Hz := _Wave_2Hz;
END_GET
END_PROPERTY

{attribute 'monitoring' := 'call'}
PROPERTY Wave_500Hz : BOOL
GET
Wave_500Hz := _Wave_500Hz;
END_GET
END_PROPERTY

{attribute 'monitoring' := 'call'}
PROPERTY Wave_50Hz : BOOL
GET
Wave_50Hz := _Wave_50Hz;
END_GET
END_PROPERTY

{attribute 'monitoring' := 'call'}
PROPERTY Wave_5Hz : BOOL
GET
Wave_5Hz := _Wave_5Hz;
END_GET
END_PROPERTY

END_FUNCTION_BLOCK

// ---- Utilities/Functions/CompareLREAL.TcPOU
FUNCTION CompareLREAL : BOOL
VAR_INPUT
	Var1	: LREAL;
	Var2	: LREAL;
	Epsilon : LREAL := 1E-6;
END_VAR

CompareLREAL := ABS(Var1 - Var2) < Epsilon;

END_FUNCTION

// ---- Utilities/Functions/CompareModulo.TcPOU
FUNCTION CompareModulo : BOOL
VAR_INPUT
	Var1	: LREAL;
	Var2	: LREAL;
	Modulo	: LREAL := 360.0;
	Epsilon : LREAL := 1E-6;
END_VAR

CompareModulo := (ABS(MODABS(Var1, Modulo) - MODABS(Var2, Modulo)) < Epsilon) OR (ABS(MODABS(Var1, Modulo) - MODABS(Var2, Modulo)) > (Modulo - Epsilon));

END_FUNCTION

// ---- Utilities/Functions/PercentToAnalog.TcPOU
FUNCTION PercentToAnalog : INT
VAR_INPUT
	TargetValue : DINT; // 0-100%
END_VAR

PercentToAnalog := TO_INT(32767 * TargetValue / 100);

END_FUNCTION

// ---- Utilities/Motion/ATAN2.TcPOU
FUNCTION ATAN2 : LREAL
VAR_INPUT
    Y : LREAL;   // Numerator   (opposite)
    X : LREAL;   // Denominator (adjacent)
END_VAR
VAR CONSTANT
    Pi     : LREAL := 3.14159265358979;
    HalfPi : LREAL := 1.57079632679490;
END_VAR

// --- Quadrant-aware arctangent, result range (-Pi .. +Pi] ---
IF X > 0.0 THEN
    // Right half-plane: direct arctangent
    ATAN2 := ATAN(Y / X);

ELSIF X < 0.0 THEN
    // Left half-plane: shift by +/- Pi depending on sign of Y
    IF Y >= 0.0 THEN
        ATAN2 := ATAN(Y / X) + Pi;
    ELSE
        ATAN2 := ATAN(Y / X) - Pi;
    END_IF

ELSE
    // X = 0: angle lies on the vertical axis
    IF Y > 0.0 THEN
        ATAN2 := HalfPi;        // +90 deg
    ELSIF Y < 0.0 THEN
        ATAN2 := -HalfPi;       // -90 deg
    ELSE
        ATAN2 := 0.0;           // Undefined (0,0) -> return 0
    END_IF
END_IF

END_FUNCTION

// ---- Utilities/Motion/CalculateHypotenuseAngle.TcPOU
FUNCTION_BLOCK CalculateHypotenuseAngle
VAR_INPUT
    a               : LREAL;   // opposite side (e.g. 0.002)
    b               : LREAL;   // adjacent side (e.g. 50)
    execute         : BOOL;
END_VAR
VAR_OUTPUT
    c               : LREAL;   // hypotenuse = SQRT(a^2 + b^2)
    angleRad        : LREAL;   // angle alpha in radians = ASIN(a / c)
    angleDeg        : LREAL;   // angle alpha in decimal degrees
END_VAR
VAR
    executeLast     : BOOL;
    degWhole        : DINT;
    degFraction     : LREAL;
    minWhole        : DINT;
    minFraction     : LREAL;
    secWhole        : DINT;
    degText         : STRING(8);
    minText         : STRING(4);
    secText         : STRING(4);
END_VAR

IF execute THEN
    c := SQRT(a * a + b * b);
 
    IF c > 0.0 THEN
        // angle alpha = ARCSIN(a / c)
        angleRad := ASIN(a / c);
        angleDeg := angleRad * 180.0 / PI;
 
        // ---- convert decimal degrees to D° M' S" ----
        degWhole    := TRUNC(angleDeg);
        degFraction := ABS(angleDeg - DINT_TO_LREAL(degWhole)) * 60.0;
 
        minWhole    := TRUNC(degFraction);
        minFraction := (degFraction - DINT_TO_LREAL(minWhole)) * 60.0;
 
        secWhole    := TRUNC(minFraction + 0.5); // round to nearest second
 
        // handle rollover from rounding (60" -> next minute, 60' -> next degree)
        IF secWhole >= 60 THEN
            secWhole := secWhole - 60;
            minWhole := minWhole + 1;
        END_IF
        IF minWhole >= 60 THEN
            minWhole := minWhole - 60;
            degWhole := degWhole + 1;
        END_IF
    ELSE
        // c = 0 -> a = b = 0, angle undefined
        angleRad := 0.0;
        angleDeg := 0.0;
    END_IF
END_IF

END_FUNCTION_BLOCK

// ---- Utilities/Motion/CalculateMotionDynamics.TcPOU
(*
    CalcMotionDynamics
    ------------------
    Calculates the "best" (= gentlest possible) set of dynamic parameters
    Velocity / Acceleration / Deceleration / Jerk so that a given distance is
    travelled in a given time, without ever exceeding the supplied maximum values.

    Method
    ------
    1) The fastest possible move for the distance is calculated using the full
       maximum dynamics. This gives TimeMin (7 phase jerk limited profile:
       jerk up - const. acceleration - jerk down - const. velocity -
       jerk up - const. deceleration - jerk down; phases collapse automatically
       when the distance or the velocity limit does not allow them).

    2) The requested time is reached by stretching exactly that profile in time.
       For a time scaling factor Lambda = TimeMin / MoveTime the identical position
       profile shape is obtained with
            v ~ Lambda, a ~ Lambda^2, j ~ Lambda^3
       This is exact: the resulting move time is TimeMin / Lambda = MoveTime, for
       every profile shape, so no iteration over the requested time is needed.

    Because the shape of the fastest profile is kept, the result is the smallest
    set of dynamics that still meets the requested time, and the utilisation of
    velocity, acceleration, deceleration and jerk stays balanced (no single value
    is driven to its limit while the others idle).

    Notes
    -----
    - JerkMax = 0 means "no jerk limitation": a trapezoidal velocity profile is
      calculated and Jerk is returned as 0.
    - Units are free but must be consistent: distance [u], time [s] =>
      velocity [u/s], acceleration/deceleration [u/s2], jerk [u/s3].
    - The model matches the standard jerk limited (trapezoidal acceleration)
      profile of TwinCAT NC PTP. If the axis is parameterised with a different
      acceleration characteristic (e.g. sin2 / smoothed), the achieved time
      deviates slightly.
    - The block is stateless, it recalculates on every call. Just call it
      cyclically (or once in a step) and read the outputs in the same cycle.
    - Very long requested times lead to very small dynamics (jerk scales with
      Lambda^3). Check ScalingFactor if the axis has a lower dynamic limit.
*)
FUNCTION_BLOCK CalculateMotionDynamics
VAR_INPUT
    /// Distance to travel [u]. The sign is ignored, ABS() is used.
    Distance : LREAL;
    /// Time in which the distance shall be travelled [s]
    MoveTime : LREAL;

    /// Maximum allowed velocity [u/s]
    VelocityMax : LREAL;
    /// Maximum allowed acceleration [u/s2]
    AccelerationMax : LREAL;
    /// Maximum allowed deceleration [u/s2]
    DecelerationMax : LREAL;
    /// Maximum allowed jerk [u/s3]. 0 = no jerk limitation.
    JerkMax : LREAL;
END_VAR
VAR_OUTPUT
    /// TRUE: outputs contain a valid dynamic set for the requested distance/time
    Valid : BOOL;
    /// TRUE: an error occurred, see ErrorId
    Error : BOOL;
    ErrorId : MotionDynamicsError;
    /// TRUE: MoveTime could not be met, the outputs contain the fastest possible profile
    TimeLimited : BOOL;

    (* --- results: feed these directly into MC_MoveAbsolute / MC_MoveRelative --- *)
    Velocity : LREAL;
    Acceleration : LREAL;
    Deceleration : LREAL;
    Jerk : LREAL;

    (* --- information --- *)
    /// Fastest possible time for Distance with the given maximum dynamics [s]
    TimeMin : LREAL;
    /// Time the calculated dynamics will actually need [s] (= MoveTime, or TimeMin if MoveTime was too short)
    TimeResulting : LREAL;
    /// Applied time scaling factor Lambda = TimeMin / MoveTime, range (0..1]
    ScalingFactor : LREAL;
    /// Highest velocity actually reached [u/s]. Lower than Velocity for short moves.
    VelocityPeak : LREAL;
    /// Duration of the acceleration phase (incl. both jerk phases) [s]
    TimeAccelerate : LREAL;
    /// Duration of the constant velocity phase [s]. 0 for short moves.
    TimeConstantVelocity : LREAL;
    /// Duration of the deceleration phase (incl. both jerk phases) [s]
    TimeDecelerate : LREAL;
END_VAR
VAR
    /// TRUE if JerkMax > 0, evaluated once per call and used by the methods
    _JerkLimited : BOOL;
    _AbsoluteDistance : LREAL;
    /// Peak velocity of the fastest profile (Lambda = 1)
    _PeakVelocityFull : LREAL;
    /// Phase times of the fastest profile (Lambda = 1)
    _TimeAccelerateFull : LREAL;
    _TimeConstantVelocityFull : LREAL;
    _TimeDecelerateFull : LREAL;
END_VAR

// ---------------------------------------------------------------- reset outputs
Valid := FALSE;
Error := FALSE;
ErrorId := MotionDynamicsError.NoError;
TimeLimited := FALSE;

Velocity := 0.0;
Acceleration := 0.0;
Deceleration := 0.0;
Jerk := 0.0;

TimeMin := 0.0;
TimeResulting := 0.0;
ScalingFactor := 0.0;
VelocityPeak := 0.0;
TimeAccelerate := 0.0;
TimeConstantVelocity := 0.0;
TimeDecelerate := 0.0;

// ------------------------------------------------------------------- validation
_AbsoluteDistance := ABS(Distance);

IF NOT (_AbsoluteDistance > 0.0) THEN
    ErrorId := MotionDynamicsError.InvalidDistance;
ELSIF NOT (MoveTime > 0.0) THEN
    ErrorId := MotionDynamicsError.InvalidMoveTime;
ELSIF NOT (VelocityMax > 0.0) THEN
    ErrorId := MotionDynamicsError.InvalidVelocityMax;
ELSIF NOT (AccelerationMax > 0.0) THEN
    ErrorId := MotionDynamicsError.InvalidAccelerationMax;
ELSIF NOT (DecelerationMax > 0.0) THEN
    ErrorId := MotionDynamicsError.InvalidDecelerationMax;
ELSIF JerkMax < 0.0 THEN
    ErrorId := MotionDynamicsError.InvalidJerkMax;
END_IF

IF ErrorId <> MotionDynamicsError.NoError THEN
    Error := TRUE;
    RETURN;
END_IF

_JerkLimited := JerkMax > 0.0;

// ------------------------------------------- fastest profile (full max dynamics)
IF _AbsoluteDistance >= AccelDecelDistance(VelocityMax) THEN
    // long move: VelocityMax is reached, a constant velocity phase exists
    _PeakVelocityFull := VelocityMax;
ELSE
    // short move: velocity limit is never reached, acceleration/jerk limit the peak
    _PeakVelocityFull := PeakVelocityForDistance(_AbsoluteDistance);

    IF NOT (_PeakVelocityFull > 0.0) OR (_PeakVelocityFull > VelocityMax * (1.0 + 1E-9)) THEN
        Error := TRUE;
        ErrorId := MotionDynamicsError.CalculationFailed;
        RETURN;
    END_IF

    // right at the boundary between short and long move the solver may return
    // VelocityMax plus a rounding error
    IF _PeakVelocityFull > VelocityMax THEN
        _PeakVelocityFull := VelocityMax;
    END_IF
END_IF

_TimeAccelerateFull := RampTime(_PeakVelocityFull, AccelerationMax);
_TimeDecelerateFull := RampTime(_PeakVelocityFull, DecelerationMax);

// distance of both ramps = PeakVelocity/2 * RampTime (velocity ramp is point symmetric)
_TimeConstantVelocityFull :=
    (_AbsoluteDistance - 0.5 * _PeakVelocityFull * (_TimeAccelerateFull + _TimeDecelerateFull))
    / _PeakVelocityFull;

IF _TimeConstantVelocityFull < 0.0 THEN
    _TimeConstantVelocityFull := 0.0;   // rounding only, the branch above guarantees >= 0
END_IF

TimeMin := _TimeAccelerateFull + _TimeConstantVelocityFull + _TimeDecelerateFull;

// --------------------------------------------------------- time scaling (Lambda)
ScalingFactor := TimeMin / MoveTime;

IF ScalingFactor > 1.0 THEN
    // requested time is faster than physically possible -> return the fastest profile
    IF ScalingFactor > (1.0 + 1E-9) THEN
        TimeLimited := TRUE;
        Error := TRUE;
        ErrorId := MotionDynamicsError.TimeTooShort;
    END_IF
    ScalingFactor := 1.0;
END_IF

// v ~ Lambda, a ~ Lambda^2, j ~ Lambda^3, times ~ 1/Lambda
Velocity := ScalingFactor * VelocityMax;
Acceleration := ScalingFactor * ScalingFactor * AccelerationMax;
Deceleration := ScalingFactor * ScalingFactor * DecelerationMax;
IF _JerkLimited THEN
    Jerk := ScalingFactor * ScalingFactor * ScalingFactor * JerkMax;
END_IF

VelocityPeak := ScalingFactor * _PeakVelocityFull;
TimeAccelerate := _TimeAccelerateFull / ScalingFactor;
TimeConstantVelocity := _TimeConstantVelocityFull / ScalingFactor;
TimeDecelerate := _TimeDecelerateFull / ScalingFactor;
TimeResulting := TimeMin / ScalingFactor;

Valid := NOT Error;

(*
    Distance needed to accelerate 0 -> TargetVelocity and decelerate back to 0
    with AccelerationMax / DecelerationMax / JerkMax.
    Strictly monotonically increasing over TargetVelocity.
*)
METHOD PRIVATE AccelDecelDistance : LREAL
VAR_INPUT
    TargetVelocity : LREAL;
END_VAR
AccelDecelDistance := 0.5 * TargetVelocity
                     * ( RampTime(TargetVelocity, AccelerationMax)
                       + RampTime(TargetVelocity, DecelerationMax) );
END_METHOD

(*
    Inverse of AccelDecelDistance(): peak velocity of a triangular move (no
    constant velocity phase) that covers exactly DistanceToTravel.
    Closed form where both ramps are in the same regime, bisection for the
    mixed case (one ramp triangular, the other trapezoidal).
*)
METHOD PRIVATE PeakVelocityForDistance : LREAL
VAR_INPUT
    DistanceToTravel : LREAL;
END_VAR
VAR
    /// velocities above which the acceleration / deceleration ramp becomes trapezoidal
    VelocityAccelerationLimit : LREAL;
    VelocityDecelerationLimit : LREAL;
    Low : LREAL;
    High : LREAL;
    Mid : LREAL;
    /// factors of QuadraticTerm*v^2 + LinearTerm*v - DistanceToTravel = 0
    QuadraticTerm : LREAL;
    LinearTerm : LREAL;
    Iteration : INT;
END_VAR
IF NOT _JerkLimited THEN
    // s = v^2/2 * (1/a + 1/d)
    PeakVelocityForDistance := SQRT(2.0 * DistanceToTravel
                                    / (1.0 / AccelerationMax + 1.0 / DecelerationMax));
    RETURN;
END_IF

VelocityAccelerationLimit := AccelerationMax * AccelerationMax / JerkMax;
VelocityDecelerationLimit := DecelerationMax * DecelerationMax / JerkMax;
Low := MIN(VelocityAccelerationLimit, VelocityDecelerationLimit);
High := MAX(VelocityAccelerationLimit, VelocityDecelerationLimit);

IF DistanceToTravel <= AccelDecelDistance(Low) THEN
    // both ramps triangular: s = 2 * v^1.5 / SQRT(j)
    PeakVelocityForDistance := EXPT(DistanceToTravel * SQRT(JerkMax) / 2.0, 2.0 / 3.0);

ELSIF DistanceToTravel >= AccelDecelDistance(High) THEN
    // both ramps trapezoidal
    QuadraticTerm := 0.5 * (1.0 / AccelerationMax + 1.0 / DecelerationMax);
    LinearTerm := 0.5 * (AccelerationMax + DecelerationMax) / JerkMax;
    PeakVelocityForDistance :=
        (-LinearTerm + SQRT(LinearTerm * LinearTerm + 4.0 * QuadraticTerm * DistanceToTravel))
        / (2.0 * QuadraticTerm);

ELSE
    // mixed regime, no closed form -> bisection on the monotonic distance function
    // (Low / High bracket the solution because of the two branches above)
    FOR Iteration := 1 TO 100 DO
        Mid := 0.5 * (Low + High);
        IF AccelDecelDistance(Mid) < DistanceToTravel THEN
            Low := Mid;
        ELSE
            High := Mid;
        END_IF
        IF (High - Low) <= (1E-12 * High) THEN
            EXIT;
        END_IF
    END_FOR
    PeakVelocityForDistance := 0.5 * (Low + High);
END_IF
END_METHOD

(*
    Duration of a velocity ramp 0 -> RampVelocity (or RampVelocity -> 0) with the
    given acceleration limit and JerkMax.
      trapezoidal acceleration (limit reached):  v/a + a/j
      triangular acceleration  (limit not hit):  2 * SQRT(v/j)
*)
METHOD PRIVATE RampTime : LREAL
VAR_INPUT
    RampVelocity : LREAL;
    AccelerationLimit : LREAL;
END_VAR
IF RampVelocity <= 0.0 THEN
    RampTime := 0.0;

ELSIF NOT _JerkLimited THEN
    RampTime := RampVelocity / AccelerationLimit;

ELSIF (RampVelocity * JerkMax) >= (AccelerationLimit * AccelerationLimit) THEN
    RampTime := RampVelocity / AccelerationLimit + AccelerationLimit / JerkMax;

ELSE
    RampTime := 2.0 * SQRT(RampVelocity / JerkMax);
END_IF
END_METHOD

END_FUNCTION_BLOCK

// ---- Utilities/Motion/CamSmoothDerivatives.TcPOU
FUNCTION_BLOCK CamSmoothDerivatives
VAR_GENERIC CONSTANT
    // Upper bound for the internal work arrays.
    // Raise if a cam table ever carries more profile points than this.
    CamMaxPoints : UINT := 53;
END_VAR
VAR_OUTPUT
    /// Reason the last Execute failed
    ErrorId : CamSmoothError;
    /// Points processed
    PointCount : INT;

    (* --- commissioning diagnostics, per master unit --- *)
    MaxSlaveVelocity : LREAL;
    MaxSlaveAcceleration : LREAL;
    MaxSlaveJerk : LREAL;
END_VAR
VAR
    _MasterPos : ARRAY[0..CamMaxPoints-1] OF LREAL;
    _SlavePos : ARRAY[0..CamMaxPoints-1] OF LREAL;
    /// Segment lengths
    _SegmentLength : ARRAY[0..CamMaxPoints-1] OF LREAL;
    /// 2nd derivatives
    _SecondDerivative : ARRAY[0..CamMaxPoints-1] OF LREAL;

    (* --- tridiagonal system over the interior unknowns _SecondDerivative[1..Count-2] --- *)
    _SubDiagonal : ARRAY[0..CamMaxPoints-1] OF LREAL;
    _Diagonal : ARRAY[0..CamMaxPoints-1] OF LREAL;
    _SuperDiagonal : ARRAY[0..CamMaxPoints-1] OF LREAL;
    _RightHandSide : ARRAY[0..CamMaxPoints-1] OF LREAL;
END_VAR

METHOD Execute : BOOL
VAR_IN_OUT
    Points : ARRAY[*] OF MC_MotionFunctionPoint;
END_VAR
VAR_INPUT
    /// Index of the first profile point to fit
    FirstIndex : DINT;
    /// Index of the last profile point to fit
    LastIndex : DINT;
    /// Number of decimals the written derivatives are rounded to, 2 -> x.xx
    Decimals : INT := 4;
    Boundary : CamSplineBoundary := CamSplineBoundary.Natural;
END_VAR
VAR
    /// Number of profile points
    Count : DINT;
    /// Number of interior unknowns, = Count - 2
    InteriorCount : DINT;
    /// Profile point index
    Index : DINT;
    /// Row of the tridiagonal system
    Row : DINT;
    Digit : INT;
    /// Elimination factor of the Thomas algorithm
    Factor : LREAL;
    /// 10^Decimals
    Scale : LREAL;
    Velocity : LREAL;
    Jerk : LREAL;
END_VAR
Execute := FALSE;
ErrorId := CamSmoothError.NoError;
PointCount := 0;
MaxSlaveVelocity := 0.0;
MaxSlaveAcceleration := 0.0;
MaxSlaveJerk := 0.0;

// ---------- validate ---------------------------------------------------
IF (Decimals < 0) OR (Decimals > 9) THEN
    ErrorId := CamSmoothError.BadDecimals;
    RETURN;
END_IF

IF     (FirstIndex < LOWER_BOUND(Points, 1))
    OR (LastIndex  > UPPER_BOUND(Points, 1))
    OR (LastIndex <= FirstIndex) THEN
    ErrorId := CamSmoothError.RangeOutsideArray;
    RETURN;
END_IF

Count := LastIndex - FirstIndex + 1;

// The not-a-knot substitution references M[2] and M[Count-3], so it needs 4 points.
IF Count < 4 THEN
    ErrorId := CamSmoothError.TooFewPoints;
    RETURN;
END_IF

IF Count > UINT_TO_DINT(CamMaxPoints) THEN
    ErrorId := CamSmoothError.TooManyPoints;
    RETURN;
END_IF

// ---------- read the master / slave columns ----------------------------
FOR Index := 0 TO Count-1 DO
    _MasterPos[Index] := Points[FirstIndex + Index].MasterPos;
    _SlavePos[Index]  := Points[FirstIndex + Index].SlavePos;
END_FOR

// MasterPos must strictly increase or the spline is undefined.
FOR Index := 0 TO Count-2 DO
    _SegmentLength[Index] := _MasterPos[Index+1] - _MasterPos[Index];
    IF _SegmentLength[Index] <= 0.0 THEN
        ErrorId := CamSmoothError.MasterNotAscending;
        RETURN;
    END_IF
END_FOR

// ---------- build the tridiagonal system -------------------------------
// Unknowns are the interior second derivatives M[1]..M[Count-2], held in rows
// 0..InteriorCount-1. M[0] and M[Count-1] are NOT unknowns - the boundary
// condition below eliminates them, which is what keeps the band strictly
// tridiagonal.
InteriorCount := Count - 2;

FOR Row := 0 TO InteriorCount-1 DO
    Index := Row + 1;
    _SubDiagonal[Row]   := _SegmentLength[Index-1];
    _Diagonal[Row]      := 2.0 * (_SegmentLength[Index-1] + _SegmentLength[Index]);
    _SuperDiagonal[Row] := _SegmentLength[Index];
    _RightHandSide[Row] := 6.0 * ( (_SlavePos[Index+1] - _SlavePos[Index]) / _SegmentLength[Index]
                                 - (_SlavePos[Index] - _SlavePos[Index-1]) / _SegmentLength[Index-1] );
END_FOR

IF Boundary = CamSplineBoundary.Natural THEN
    // M[0] = M[Count-1] = 0, so their coefficients simply drop out.
    _SubDiagonal[0]                 := 0.0;
    _SuperDiagonal[InteriorCount-1] := 0.0;
ELSE
    // Not-a-knot: segments 0 and 1 are one cubic, so M is linear across
    // x[0..2]   ->   M[0] = M[1] + (M[1] - M[2]) * h[0]/h[1].
    // Substituting that into row 0 folds M[0] away. Mirrored at the far end.
    // Note: folding the raw not-a-knot row into the band instead would give
    // _Diagonal[0] = 0 for uniform spacing and kill the Thomas pivot.
    _SubDiagonal[0]   := 0.0;
    _Diagonal[0]      := 3.0*_SegmentLength[0] + 2.0*_SegmentLength[1]
                         + _SegmentLength[0]*_SegmentLength[0]/_SegmentLength[1];
    _SuperDiagonal[0] := _SegmentLength[1] - _SegmentLength[0]*_SegmentLength[0]/_SegmentLength[1];

    _SuperDiagonal[InteriorCount-1] := 0.0;
    _Diagonal[InteriorCount-1]      := 2.0*_SegmentLength[Count-3] + 3.0*_SegmentLength[Count-2]
                                       + _SegmentLength[Count-2]*_SegmentLength[Count-2]/_SegmentLength[Count-3];
    _SubDiagonal[InteriorCount-1]   := _SegmentLength[Count-3]
                                       - _SegmentLength[Count-2]*_SegmentLength[Count-2]/_SegmentLength[Count-3];
END_IF

// ---------- Thomas algorithm -------------------------------------------
FOR Row := 1 TO InteriorCount-1 DO
    IF ABS(_Diagonal[Row-1]) < 1.0E-30 THEN
        ErrorId := CamSmoothError.SolverSingular;
        RETURN;
    END_IF
    Factor              := _SubDiagonal[Row] / _Diagonal[Row-1];
    _Diagonal[Row]      := _Diagonal[Row] - Factor * _SuperDiagonal[Row-1];
    _RightHandSide[Row] := _RightHandSide[Row] - Factor * _RightHandSide[Row-1];
END_FOR

IF ABS(_Diagonal[InteriorCount-1]) < 1.0E-30 THEN
    ErrorId := CamSmoothError.SolverSingular;
    RETURN;
END_IF

// row Row holds M[Row+1]
_SecondDerivative[InteriorCount] := _RightHandSide[InteriorCount-1] / _Diagonal[InteriorCount-1];
FOR Row := InteriorCount-2 TO 0 BY -1 DO
    _SecondDerivative[Row+1] := (_RightHandSide[Row] - _SuperDiagonal[Row] * _SecondDerivative[Row+2])
                                / _Diagonal[Row];
END_FOR

// ---------- recover the two end values ---------------------------------
IF Boundary = CamSplineBoundary.Natural THEN
    _SecondDerivative[0]       := 0.0;
    _SecondDerivative[Count-1] := 0.0;
ELSE
    _SecondDerivative[0]       := _SecondDerivative[1]
                                  + (_SecondDerivative[1] - _SecondDerivative[2])
                                    * _SegmentLength[0] / _SegmentLength[1];
    _SecondDerivative[Count-1] := _SecondDerivative[Count-2]
                                  + (_SecondDerivative[Count-2] - _SecondDerivative[Count-3])
                                    * _SegmentLength[Count-2] / _SegmentLength[Count-3];
END_IF

// ---------- write the derivatives back ---------------------------------
Scale := 1.0;
FOR Digit := 1 TO Decimals DO
    Scale := Scale * 10.0;
END_FOR

FOR Index := 0 TO Count-1 DO
    IF Index < Count-1 THEN
        Velocity := (_SlavePos[Index+1] - _SlavePos[Index]) / _SegmentLength[Index]
                    - _SegmentLength[Index] * (2.0*_SecondDerivative[Index] + _SecondDerivative[Index+1]) / 6.0;
        Jerk     := (_SecondDerivative[Index+1] - _SecondDerivative[Index]) / _SegmentLength[Index];
    ELSE
        // last point: evaluate the previous segment at its far end
        Velocity := (_SlavePos[Count-1] - _SlavePos[Count-2]) / _SegmentLength[Count-2]
                    + _SegmentLength[Count-2] * (_SecondDerivative[Count-2] + 2.0*_SecondDerivative[Count-1]) / 6.0;
        Jerk     := (_SecondDerivative[Count-1] - _SecondDerivative[Count-2]) / _SegmentLength[Count-2];
    END_IF

    Points[FirstIndex + Index].SlaveVelo := RoundTo(Velocity, Scale);
    Points[FirstIndex + Index].SlaveAcc  := RoundTo(_SecondDerivative[Index], Scale);
    Points[FirstIndex + Index].SlaveJerk := RoundTo(Jerk, Scale);

    MaxSlaveVelocity     := MAX(MaxSlaveVelocity,     ABS(Points[FirstIndex + Index].SlaveVelo));
    MaxSlaveAcceleration := MAX(MaxSlaveAcceleration, ABS(Points[FirstIndex + Index].SlaveAcc));
    MaxSlaveJerk         := MAX(MaxSlaveJerk,         ABS(Points[FirstIndex + Index].SlaveJerk));
END_FOR

PointCount := DINT_TO_INT(Count);
Execute := TRUE;
END_METHOD

METHOD RoundTo : LREAL
VAR_INPUT
    Value : LREAL;
    /// 10^Decimals
    Scale : LREAL;
END_VAR
// LREAL_TO_LINT rounds to the nearest integer under IEC 61131-3 conversion
// semantics, so no explicit +/- 0.5 is needed. Any realistic cam derivative
// scaled by 10^9 stays far inside the LINT range. Also normalises -0.0 to 0.0.
RoundTo := LINT_TO_LREAL( LREAL_TO_LINT( Value * Scale ) ) / Scale;
END_METHOD

END_FUNCTION_BLOCK

// ---- Utilities/Motion/XPlanar6DMoverToWorldTransform.TcPOU
(* ============================================================================
   FUNCTION BLOCK: FB_MoverToWorldTransform
   ----------------------------------------------------------------------------
   PURPOSE:
     Forward transforms a mover tooling position from the mover (local) frame
     into the world coordinate system of the tile.

     Coordinate chain:
       World (Tile) <-- Mover Pose <-- Tool Offset <-- Tool Tip

     Rotation convention: INTRINSIC XYZ (Tait-Bryan)
       Rx applied first (roll around X), then Ry (pitch around Y'),
       then Rz (yaw around Z'').
       Combined matrix: R = Rz * Ry * Rx

     Runs every scan cycle — no enable trigger required.
     All output angles are ABSOLUTE (unbounded, no rollover).

   INPUTS:
     MoverX, MoverY, MoverZ          : Mover position in tile world [mm]
     MoverRx, MoverRy, MoverRz       : Mover orientation in tile world [°]
                                       XYZ intrinsic: Rx first, Rz last
     ToolOffsetX/Y/Z                 : Tool offset in mover-local frame [mm]
     ToolOffsetRx/Ry/Rz             : Tool orientation offset in mover frame [°]
     Reset                           : Clears accumulated angle unwrap history

   OUTPUTS:
     WorldX, WorldY, WorldZ          : Tool tip position in tile world [mm]
     WorldRx, WorldRy, WorldRz       : Tool tip orientation in tile world [°]
                                       ABSOLUTE — never rolls over ±360°
     Error                           : Set TRUE when asin clamp fires (near ±90° pitch)
   ============================================================================ *)

FUNCTION_BLOCK XPlanar6DMoverToWorldTransform
VAR_INPUT
    MoverX          : LREAL;
    MoverY          : LREAL;
    MoverZ          : LREAL;
    MoverRx         : LREAL;   (* Roll  around X [°] — applied first  *)
    MoverRy         : LREAL;   (* Pitch around Y [°] — applied second *)
    MoverRz         : LREAL;   (* Yaw   around Z [°] — applied last   *)

    ToolOffsetX     : LREAL;
    ToolOffsetY     : LREAL;
    ToolOffsetZ     : LREAL;
    ToolOffsetRx    : LREAL;
    ToolOffsetRy    : LREAL;
    ToolOffsetRz    : LREAL;

    Reset           : BOOL;
END_VAR

VAR_OUTPUT
    WorldX          : LREAL;
    WorldY          : LREAL;
    WorldZ          : LREAL;
    WorldRx         : LREAL;   (* Absolute, no rollover *)
    WorldRy         : LREAL;   (* Absolute, no rollover *)
    WorldRz         : LREAL;   (* Absolute, no rollover *)
    Error           : BOOL;
END_VAR

VAR
    ResetPrev       : BOOL;

    R_M             : ARRAY[1..3, 1..3] OF LREAL;   (* Mover rotation matrix    *)
    R_T             : ARRAY[1..3, 1..3] OF LREAL;   (* Tool offset rot. matrix  *)
    R_W             : ARRAY[1..3, 1..3] OF LREAL;   (* Combined world rot. matrix *)

    Dx              : LREAL;   (* Tool offset rotated into world frame *)
    Dy              : LREAL;
    Dz              : LREAL;

    RawRx           : LREAL;   (* Wrapped angles extracted from R_W *)
    RawRy           : LREAL;
    RawRz           : LREAL;

    PrevRawRx       : LREAL;
    PrevRawRy       : LREAL;
    PrevRawRz       : LREAL;

    UnwrapOffRx     : LREAL;   (* Accumulated unwrap corrections *)
    UnwrapOffRy     : LREAL;
    UnwrapOffRz     : LREAL;

    FirstCalc       : BOOL := TRUE;

    Cx              : LREAL;   (* Trig intermediates — mover *)
    Sx              : LREAL;
    Cy              : LREAL;
    Sy              : LREAL;
    Cz              : LREAL;
    Sz              : LREAL;

    Cx2             : LREAL;   (* Trig intermediates — tool offset *)
    Sx2             : LREAL;
    Cy2             : LREAL;
    Sy2             : LREAL;
    Cz2             : LREAL;
    Sz2             : LREAL;

    SyWorld         : LREAL;   (* Clamped sin(Ry_world) for gimbal guard *)
END_VAR

VAR CONSTANT
    DEG2RAD         : LREAL := 0.017453292519943295;
    RAD2DEG         : LREAL := 57.29577951308232;
    HALF_TURN       : LREAL := 180.0;
    FULL_TURN       : LREAL := 360.0;
END_VAR

(* ── Reset unwrap history on rising edge ────────────────────────────────────── *)
IF Reset AND NOT ResetPrev THEN
    UnwrapOffRx := 0.0;
    UnwrapOffRy := 0.0;
    UnwrapOffRz := 0.0;
    PrevRawRx   := 0.0;
    PrevRawRy   := 0.0;
    PrevRawRz   := 0.0;
    FirstCalc   := TRUE;
    Error       := FALSE;
END_IF
ResetPrev := Reset;

Error := FALSE;

(* ============================================================================
   MOVER ROTATION MATRIX  R_M = Rz(MoverRz) * Ry(MoverRy) * Rx(MoverRx)
   ============================================================================ *)
Cx := COS(MoverRx * DEG2RAD);
Sx := SIN(MoverRx * DEG2RAD);
Cy := COS(MoverRy * DEG2RAD);
Sy := SIN(MoverRy * DEG2RAD);
Cz := COS(MoverRz * DEG2RAD);
Sz := SIN(MoverRz * DEG2RAD);

R_M[1,1] :=  Cy * Cz;
R_M[1,2] :=  Sx * Sy * Cz - Cx * Sz;
R_M[1,3] :=  Cx * Sy * Cz + Sx * Sz;

R_M[2,1] :=  Cy * Sz;
R_M[2,2] :=  Sx * Sy * Sz + Cx * Cz;
R_M[2,3] :=  Cx * Sy * Sz - Sx * Cz;

R_M[3,1] := -Sy;
R_M[3,2] :=  Sx * Cy;
R_M[3,3] :=  Cx * Cy;

(* ============================================================================
   TOOL OFFSET ROTATION MATRIX  R_T = Rz(ToolOffsetRz) * Ry(ToolOffsetRy) * Rx(ToolOffsetRx)
   ============================================================================ *)
Cx2 := COS(ToolOffsetRx * DEG2RAD);
Sx2 := SIN(ToolOffsetRx * DEG2RAD);
Cy2 := COS(ToolOffsetRy * DEG2RAD);
Sy2 := SIN(ToolOffsetRy * DEG2RAD);
Cz2 := COS(ToolOffsetRz * DEG2RAD);
Sz2 := SIN(ToolOffsetRz * DEG2RAD);

R_T[1,1] :=  Cy2 * Cz2;
R_T[1,2] :=  Sx2 * Sy2 * Cz2 - Cx2 * Sz2;
R_T[1,3] :=  Cx2 * Sy2 * Cz2 + Sx2 * Sz2;

R_T[2,1] :=  Cy2 * Sz2;
R_T[2,2] :=  Sx2 * Sy2 * Sz2 + Cx2 * Cz2;
R_T[2,3] :=  Cx2 * Sy2 * Sz2 - Sx2 * Cz2;

R_T[3,1] := -Sy2;
R_T[3,2] :=  Sx2 * Cy2;
R_T[3,3] :=  Cx2 * Cy2;

(* ============================================================================
   COMBINED WORLD ROTATION  R_W = R_M * R_T
   ============================================================================ *)
R_W[1,1] := R_M[1,1]*R_T[1,1] + R_M[1,2]*R_T[2,1] + R_M[1,3]*R_T[3,1];
R_W[1,2] := R_M[1,1]*R_T[1,2] + R_M[1,2]*R_T[2,2] + R_M[1,3]*R_T[3,2];
R_W[1,3] := R_M[1,1]*R_T[1,3] + R_M[1,2]*R_T[2,3] + R_M[1,3]*R_T[3,3];

R_W[2,1] := R_M[2,1]*R_T[1,1] + R_M[2,2]*R_T[2,1] + R_M[2,3]*R_T[3,1];
R_W[2,2] := R_M[2,1]*R_T[1,2] + R_M[2,2]*R_T[2,2] + R_M[2,3]*R_T[3,2];
R_W[2,3] := R_M[2,1]*R_T[1,3] + R_M[2,2]*R_T[2,3] + R_M[2,3]*R_T[3,3];

R_W[3,1] := R_M[3,1]*R_T[1,1] + R_M[3,2]*R_T[2,1] + R_M[3,3]*R_T[3,1];
R_W[3,2] := R_M[3,1]*R_T[1,2] + R_M[3,2]*R_T[2,2] + R_M[3,3]*R_T[3,2];
R_W[3,3] := R_M[3,1]*R_T[1,3] + R_M[3,2]*R_T[2,3] + R_M[3,3]*R_T[3,3];

(* ============================================================================
   WORLD POSITION
   Tool offset translated by R_M into the world frame, added to mover position
   ============================================================================ *)
Dx := R_M[1,1]*ToolOffsetX + R_M[1,2]*ToolOffsetY + R_M[1,3]*ToolOffsetZ;
Dy := R_M[2,1]*ToolOffsetX + R_M[2,2]*ToolOffsetY + R_M[2,3]*ToolOffsetZ;
Dz := R_M[3,1]*ToolOffsetX + R_M[3,2]*ToolOffsetY + R_M[3,3]*ToolOffsetZ;

WorldX := MoverX + Dx;
WorldY := MoverY + Dy;
WorldZ := MoverZ + Dz;

(* ============================================================================
   EXTRACT XYZ EULER ANGLES FROM R_W
     Ry = asin( -R_W[3,1] )
     Rx = atan2(  R_W[3,2],  R_W[3,3] )
     Rz = atan2(  R_W[2,1],  R_W[1,1] )
   R_W[3,1] clamped to [-1, 1] to prevent NaN at the ±90° pitch singularity
   ============================================================================ *)
SyWorld := R_W[3,1];
IF SyWorld >  1.0 THEN SyWorld :=  1.0; Error := TRUE; END_IF
IF SyWorld < -1.0 THEN SyWorld := -1.0; Error := TRUE; END_IF

RawRy := ASIN(-SyWorld)            * RAD2DEG;
RawRx := ATAN2(R_W[3,2], R_W[3,3]) * RAD2DEG;
RawRz := ATAN2(R_W[2,1], R_W[1,1]) * RAD2DEG;

(* ============================================================================
   ANGLE UNWRAP — prevent ±360° rollover
   ASIN output is bounded to [-90, +90] and ATAN2 to [-180, +180], so a raw
   angle can jump at most 360° per cycle. A single IF per axis is sufficient.
   ============================================================================ *)
IF FirstCalc THEN
    PrevRawRx   := RawRx;
    PrevRawRy   := RawRy;
    PrevRawRz   := RawRz;
    UnwrapOffRx := 0.0;
    UnwrapOffRy := 0.0;
    UnwrapOffRz := 0.0;
    FirstCalc   := FALSE;
ELSE
    IF (RawRx - PrevRawRx) >  HALF_TURN THEN UnwrapOffRx := UnwrapOffRx - FULL_TURN; END_IF
    IF (RawRx - PrevRawRx) < -HALF_TURN THEN UnwrapOffRx := UnwrapOffRx + FULL_TURN; END_IF

    IF (RawRy - PrevRawRy) >  HALF_TURN THEN UnwrapOffRy := UnwrapOffRy - FULL_TURN; END_IF
    IF (RawRy - PrevRawRy) < -HALF_TURN THEN UnwrapOffRy := UnwrapOffRy + FULL_TURN; END_IF

    IF (RawRz - PrevRawRz) >  HALF_TURN THEN UnwrapOffRz := UnwrapOffRz - FULL_TURN; END_IF
    IF (RawRz - PrevRawRz) < -HALF_TURN THEN UnwrapOffRz := UnwrapOffRz + FULL_TURN; END_IF

    PrevRawRx := RawRx;
    PrevRawRy := RawRy;
    PrevRawRz := RawRz;
END_IF

(* ── Absolute output angles ─────────────────────────────────────────────────── *)
WorldRx := RawRx + UnwrapOffRx;
WorldRy := RawRy + UnwrapOffRy;
WorldRz := RawRz + UnwrapOffRz;

END_FUNCTION_BLOCK

// ---- Utilities/Timing/Stopwatch.TcPOU
FUNCTION_BLOCK Stopwatch
VAR
	StartTime			: T_DCTIME64;
	EndTime				: T_DCTIME64;
	PreviousLapEndTime	: T_DCTIME64;
	PreviousElapsedTime : LREAL;
	_Running			: BOOL;
END_VAR

VAR CONSTANT
	OneNanosecond : LREAL := 1.0E-9;
END_VAR

{attribute 'monitoring' := 'call'}
PROPERTY Elapsed : LREAL
GET
IF _Running THEN
	Elapsed := TO_LREAL(F_GetCurDcTickTime64() - StartTime) * OneNanosecond;
ELSE
	Elapsed := PreviousElapsedTime;
END_IF
END_GET
END_PROPERTY

METHOD Lap : LREAL;
VAR
	LapEndTime	: T_DCTIME64;
	LapDuration : LREAL;
END_VAR
IF _Running THEN
	LapEndTime		   := F_GetActualDcTime64();
	LapDuration		   := TO_LREAL(LapEndTime - PreviousLapEndTime) * OneNanosecond;
	PreviousLapEndTime := LapEndTime;
	Lap				   := LapDuration;
END_IF
END_METHOD

{attribute 'monitoring' := 'call'}
PROPERTY Running : BOOL
GET
Running := _Running;
END_GET
END_PROPERTY

METHOD Start
StartTime			:= F_GetActualDcTime64();
PreviousLapEndTime	:= StartTime;
_Running			:= TRUE;
PreviousElapsedTime := 0.0;
PreviousElapsedTime := 0;
END_METHOD

METHOD Stop : LREAL
IF _Running THEN
	EndTime				:= F_GetActualDcTime64();
	_Running			:= FALSE;
	PreviousElapsedTime := TO_LREAL(EndTime - StartTime) * OneNanosecond;
	Stop				:= PreviousElapsedTime;
ELSE
	Stop := 0.0;
END_IF
END_METHOD

END_FUNCTION_BLOCK

// ---- Visitors/Enable/CheckComponentsEnabledVisitor.TcPOU
FUNCTION_BLOCK CheckComponentsEnabledVisitor IMPLEMENTS I_ComponentVisitor
VAR
	Enablable : I_Enablable;
	_Enabled  : BOOL;
END_VAR

METHOD Check
VAR_INPUT
	Components : I_ComponentCollection;
END_VAR
_Enabled := TRUE;
Components.Accept(THIS^);
END_METHOD

{attribute 'monitoring' := 'call'}
PROPERTY Enabled : BOOL
GET
Enabled := _Enabled;
END_GET
END_PROPERTY

METHOD VisitComponent
VAR_INPUT
	Component : I_Component;
END_VAR
IF __QUERYINTERFACE(Component, Enablable) THEN
	IF NOT Enablable.Enabled THEN
		_Enabled := FALSE;
	END_IF
END_IF
END_METHOD

END_FUNCTION_BLOCK

// ---- Visitors/Enable/DisableAllComponentsVisitor.TcPOU
FUNCTION_BLOCK DisableAllComponentsVisitor IMPLEMENTS I_ComponentVisitor
VAR
	Enablable : I_Enablable;
	_Enabled  : BOOL;
END_VAR

METHOD Disable
VAR_INPUT
	Components : I_ComponentCollection;
END_VAR
_Enabled := FALSE;
Components.Accept(THIS^);
END_METHOD

{attribute 'monitoring' := 'call'}
PROPERTY Enabled : BOOL
GET
Enabled := _Enabled;
END_GET
END_PROPERTY

METHOD VisitComponent
VAR_INPUT
	Component : I_Component;
END_VAR
IF __QUERYINTERFACE(Component, Enablable) THEN
	Enablable.Disable();
	IF Enablable.Enabled THEN
		_Enabled := TRUE;
	END_IF
END_IF
END_METHOD

END_FUNCTION_BLOCK

// ---- Visitors/Enable/EnableAllComponentsVisitor.TcPOU
FUNCTION_BLOCK EnableAllComponentsVisitor IMPLEMENTS I_ComponentVisitor
VAR
	Enablable	   : I_Enablable;
	_Enabled	   : BOOL;
	ErrorComponent : I_Component;
END_VAR

METHOD Enable
VAR_INPUT
	Components : I_ComponentCollection;
END_VAR
_Enabled := TRUE;
Components.Accept(THIS^);
END_METHOD

{attribute 'monitoring' := 'call'}
PROPERTY Enabled : BOOL
GET
Enabled := _Enabled;
END_GET
END_PROPERTY

METHOD VisitComponent
VAR_INPUT
	Component : I_Component;
END_VAR
IF __QUERYINTERFACE(Component, Enablable) THEN
	Enablable.Enable();
	IF NOT Enablable.Enabled THEN
		ErrorComponent := Component;
		_Enabled	   := FALSE;
	END_IF
END_IF
END_METHOD

END_FUNCTION_BLOCK

// ---- Visitors/Events/GetActiveEventSeverityVisitor.TcPOU
FUNCTION_BLOCK GetActiveEventSeverityVisitor IMPLEMENTS I_ModuleVisitor, I_ComponentVisitor
VAR
	EntryModule			 : I_Module;
	HighestEventSeverity : TcEventSeverity;
	TcEventClass		 : I_EventClassTcEvents;
END_VAR

PROPERTY ActiveEventSeverity : TcEventSeverity
GET
HighestEventSeverity := Global.TcEventSeverity.Verbose;
EntryModule.Accept(THIS^);
ActiveEventSeverity := HighestEventSeverity;
END_GET
END_PROPERTY

(*FB_Init is always available implicitly and it is used primarily for initialization.
The return value is not evaluated. For a specific influence, you can also declare the
methods explicitly and provide additional code there with the standard initialization
code. You can evaluate the return value.*)
METHOD FB_Init : BOOL
VAR_INPUT
	(* TRUE: the retain variables are initialized (reset warm / reset cold)*)
	bInitRetains : BOOL;

	(* TRUE: the instance will be copied to the copy code afterward (online change)   *)
	bInCopyCode : BOOL;
	EntryModule : I_Module;
END_VAR
THIS^.EntryModule := EntryModule;
END_METHOD

METHOD VisitComponent
VAR_INPUT
	Component : I_Component;
END_VAR

VAR
	Severity : TcEventSeverity;
END_VAR
IF __QUERYINTERFACE(Component, TcEventClass) THEN
	Severity := TcEventClass.GetHighestActiveEventSeverity();
	IF Severity > HighestEventSeverity THEN
		HighestEventSeverity := Severity;
	END_IF
END_IF
END_METHOD

METHOD VisitModule
VAR_INPUT
	Module : I_Module;
END_VAR

VAR
	Severity : TcEventSeverity;
END_VAR
Module.Components.Accept(THIS^);
Module.Modules.Accept(THIS^);
IF __QUERYINTERFACE(Module, TcEventClass) THEN
	Severity := TcEventClass.GetHighestActiveEventSeverity();
	IF Severity > HighestEventSeverity THEN
		HighestEventSeverity := Severity;
	END_IF
END_IF
END_METHOD

END_FUNCTION_BLOCK

// ---- Visitors/HMI/GetSystemTreeJsonHmiVisitor.TcPOU
FUNCTION_BLOCK GetSystemTreeJsonHmiVisitor
VAR_GENERIC CONSTANT
	TreeMax : UDINT := 10000;
END_VAR IMPLEMENTS I_ModuleVisitor, I_ComponentVisitor
VAR
	{ attribute 'TcHmiSymbol.AddSymbol' }
	{ attribute 'TcHmiSymbol.AddSymbol.UserGroups' := '__SystemAdministrators,Admin' }
	SystemHmiTree : STRING(TreeMax);
	{attribute 'hide'}
	Module : I_Module;
	{attribute 'hide'}
	HmiFunction : I_HmiFunction;
	{attribute 'hide'}
	Json : FB_JsonSaxWriter;
	{attribute 'hide'}
	Entry	 : T_MaxString;
	LinkRoot : STRING;
END_VAR

METHOD PRIVATE Clear
VAR_INPUT
END_VAR
MEMSET(ADR(SystemHmiTree), 0, SIZEOF(SystemHmiTree));
Json.ResetDocument();
END_METHOD

//FB_Init is always available implicitly and it is used primarily for initialization.

//The return value is not evaluated. For a specific influence, you can also declare the

//methods explicitly and provide additional code there with the standard initialization

//code. You can evaluate the return value.
METHOD FB_Init : BOOL
VAR_INPUT
	bInitRetains : BOOL; // TRUE: the retain variables are initialized (reset warm / reset cold)
	bInCopyCode	 : BOOL; // TRUE: the instance will be copied to the copy code afterward (online change)   
	LinkRoot	 : STRING;
END_VAR
THIS^.LinkRoot := LinkRoot;
END_METHOD

METHOD GetTree
VAR_INPUT
	EntryModule : I_Module;
END_VAR
IF EntryModule = 0 THEN
	RETURN;
END_IF

Module := EntryModule;
Clear();
Json.StartObject();
Entry := Module.Name;
Json.AddKey(Entry);
Json.StartArray();
Module.Components.Accept(THIS^);
Json.EndArray();
Module.Modules.Accept(THIS^);
Json.EndObject();
Json.CopyDocument(pDoc := SystemHmiTree, nDoc := SIZEOF(SystemHmiTree));
END_METHOD

METHOD VisitComponent
VAR_INPUT
	Component : I_Component;
END_VAR
IF __QUERYINTERFACE(Component, HmiFunction) THEN
	Json.StartObject();
	Entry := HmiFunction.ControlType;
	Json.AddKeyString('ControlType', Entry);
	Entry := RIGHT(HmiFunction.InstancePath, (LEN(HmiFunction.InstancePath) - FIND(HmiFunction.InstancePath, LinkRoot)) + 1);
	Entry := CONCAT(CONCAT(Entry, '.'), HmiFunction.LinkObject);
	Json.AddKeyString('LinkPath', Entry);
	Json.EndObject();
END_IF
END_METHOD

METHOD VisitModule
VAR_INPUT
	Module : I_Module;
END_VAR
Entry := Module.Name;
IF Entry <> '' THEN
	Json.AddKey(Entry);
	Json.StartArray();
	Module.Components.Accept(THIS^);
	Json.EndArray();
	Module.Modules.Accept(THIS^);
END_IF
END_METHOD

END_FUNCTION_BLOCK

// ---- Visitors/HMI/HmiEnableDisableAllVisitor.TcPOU
FUNCTION_BLOCK HmiEnableDisableAllVisitor IMPLEMENTS I_ComponentVisitor, I_ModuleVisitor
VAR
	{attribute 'hide'}
	HmiFunction : I_HmiFunction;
	{attribute 'hide'}
	Enable : BOOL;
END_VAR

METHOD DisableHmi
VAR_INPUT
	Module : I_Module;
END_VAR
Enable := FALSE;
Module.Accept(THIS^);
END_METHOD

METHOD EnableHmi
VAR_INPUT
	Module : I_Module;
END_VAR
Enable := TRUE;
Module.Accept(THIS^);
END_METHOD

METHOD VisitComponent
VAR_INPUT
	Component : I_Component;
END_VAR
IF __QUERYINTERFACE(Component, HmiFunction) THEN
	IF Enable THEN
		HmiFunction.Enable();
	ELSE
		HmiFunction.Disable();
	END_IF
END_IF
END_METHOD

METHOD VisitModule
VAR_INPUT
	Module : I_Module;
END_VAR
Module.Components.Accept(THIS^);
Module.Modules.Accept(THIS^);
END_METHOD

END_FUNCTION_BLOCK

// ---- Visitors/Override/SetAllOverrideVisitor.TcPOU
FUNCTION_BLOCK SetAllOverrideVisitor IMPLEMENTS I_ModuleVisitor, I_ComponentVisitor
VAR
	ipOverride : I_Override;
	_Override  : LREAL;
END_VAR

METHOD Set
VAR_INPUT
	Module	 : I_Module;
	Override : LREAL;
END_VAR
_Override := Override;
Module.Accept(THIS^);
IF __QUERYINTERFACE(Module, ipOverride) THEN
	ipOverride.Override := _Override;
END_IF
END_METHOD

METHOD VisitComponent
VAR_INPUT
	Component : I_Component;
END_VAR
IF __QUERYINTERFACE(Component, ipOverride) THEN
	ipOverride.Override := _Override;
END_IF
END_METHOD

METHOD VisitModule
VAR_INPUT
	Module : I_Module;
END_VAR
Module.Components.Accept(THIS^);
Module.Modules.Accept(THIS^);
IF __QUERYINTERFACE(Module, ipOverride) THEN
	ipOverride.Override := _Override;
END_IF
END_METHOD

END_FUNCTION_BLOCK

// ---- Visitors/PackML Statemachine/ChangePackMLStateOnAllSubModulesVisitor.TcPOU
FUNCTION_BLOCK ChangePackMLStateOnAllSubModulesVisitor IMPLEMENTS I_ModuleVisitor
VAR
	PackMLCommand : E_PMLCommand;
	Statemachine  : I_ContainStatemachine;
	StateChanged  : BOOL;
	CheckState	  : E_PMLState;
END_VAR

METHOD ChangeState : BOOL;
VAR_INPUT
	PackMLCommand : E_PMLCommand;
	Module		  : I_Module;
END_VAR
StateChanged		:= TRUE;
THIS^.PackMLCommand := PackMLCommand;
CASE THIS^.PackMLCommand OF
	E_PMLCommand.Abort:
		CheckState := E_PMLState.Aborted;

	E_PMLCommand.Clear, E_PMLCommand.Stop:
		CheckState := E_PMLState.Stopped;

	E_PMLCommand.Complete:
		CheckState := E_PMLState.Completed;

	E_PMLCommand.Hold:
		CheckState := E_PMLState.Held;

	E_PMLCommand.Reset:
		CheckState := E_PMLState.Idle;

	E_PMLCommand.Start, E_PMLCommand.Unhold, E_PMLCommand.Unsuspend:
		CheckState := E_PMLState.Execute;

	E_PMLCommand.Suspend:
		CheckState := E_PMLState.Suspended;

	E_PMLCommand.Undefined:
		CheckState := E_PMLState.Undefined;
END_CASE

Module.Modules.Accept(THIS^);
ChangeState := StateChanged;
END_METHOD

METHOD VisitModule
VAR_INPUT
	Module : I_Module;
END_VAR

VAR_INST
	ReturnModule : I_Module;
END_VAR
IF __QUERYINTERFACE(Module, Statemachine) THEN
	IF Statemachine.Statemachine = 0 THEN
		ReturnModule := Module;
		RETURN;
	END_IF

	Statemachine.Statemachine.ChangeState(THIS^.PackMLCommand);
	IF Statemachine.Statemachine.CurrentState <> CheckState THEN
		StateChanged := FALSE;
	END_IF
END_IF
END_METHOD

END_FUNCTION_BLOCK

// ---- Visitors/PackML Statemachine/EventReactorPackMLVisitor.TcPOU
FUNCTION_BLOCK EventReactorPackMLVisitor EXTENDS CyclicComponent IMPLEMENTS I_ModuleVisitor, I_ComponentVisitor
VAR
	EntryModule			 : I_Module;
	HighestEventReaction : DINT;
	EventReaction		 : I_EventReaction;
	ModuleStatemachine	 : I_ContainStatemachine;
	ReactedName			 : T_MaxString;
END_VAR

METHOD CyclicLogic
IF ModuleStatemachine = 0 THEN
	RETURN;
END_IF

HighestEventReaction := 0;
EntryModule.Accept(THIS^);
CASE HighestEventReaction OF
	0:	  // Verbose
	1:	  // Info
	2:	  // Warning
	3, 4: // Error & Critical
		IF ModuleStatemachine.Statemachine.CurrentState <> E_PMLState.Aborted AND ModuleStatemachine.Statemachine.CurrentState <> E_PMLState.Aborting AND ModuleStatemachine.Statemachine.CurrentState <> E_PMLState.Clearing THEN
			Trace.LogMessage('Module or Component leading to reaction', ReactedName);
			ModuleStatemachine.Statemachine.ChangeState(E_PMLCommand.Abort);
			ReactedName := '';
		END_IF
END_CASE
END_METHOD

(*FB_Init is always available implicitly and it is used primarily for initialization.
The return value is not evaluated. For a specific influence, you can also declare the
methods explicitly and provide additional code there with the standard initialization
code. You can evaluate the return value.*)
METHOD FB_Init : BOOL
VAR_INPUT
	(* TRUE: the retain variables are initialized (reset warm / reset cold)*)
	bInitRetains : BOOL;

	(* TRUE: the instance will be copied to the copy code afterward (online change)   *)
	bInCopyCode : BOOL;
	Name		: T_MaxString;
	EntryModule : I_Module;
END_VAR
THIS^.EntryModule := EntryModule;
__QUERYINTERFACE(EntryModule, ModuleStatemachine);
END_METHOD

METHOD VisitComponent
VAR_INPUT
	Component : I_Component;
END_VAR

VAR
	Reaction : DINT;
END_VAR
IF __QUERYINTERFACE(Component, EventReaction) THEN
	Reaction := EventReaction.GetHighestActiveEventReaction();
	IF Reaction > HighestEventReaction THEN
		IF ReactedName = '' THEN
			ReactedName := Component.Name;
		END_IF

		HighestEventReaction := Reaction;
	END_IF
END_IF
END_METHOD

METHOD VisitModule
VAR_INPUT
	Module : I_Module;
END_VAR

VAR
	Reaction : DINT;
END_VAR
Module.Components.Accept(THIS^);
Module.Modules.Accept(THIS^);
IF __QUERYINTERFACE(Module, EventReaction) THEN
	Reaction := EventReaction.GetHighestActiveEventReaction();
	IF Reaction > HighestEventReaction THEN
		IF ReactedName = '' THEN
			ReactedName := Module.Name;
		END_IF

		HighestEventReaction := Reaction;
	END_IF
END_IF
END_METHOD

END_FUNCTION_BLOCK

// ---- Visitors/Reset/ResetAllVisitor.TcPOU
FUNCTION_BLOCK ResetAllVisitor IMPLEMENTS I_ModuleVisitor, I_ComponentVisitor, I_TaskResult
VAR
	{attribute 'hide'}
	Resettable : I_Resettable;
	{attribute 'hide'}
	Result : I_TaskResult;
	{attribute 'hide'}
	_Busy : BOOL;
	{attribute 'hide'}
	_Error : BOOL;
	{attribute 'hide'}
	_ErrorId	   : UDINT;
	ErrorComponent : I_Component;
	ErrorModule	   : I_Module;
END_VAR

{attribute 'monitoring' := 'call'}
PROPERTY Busy : BOOL
GET
Busy := _Busy;
END_GET
END_PROPERTY

{attribute 'monitoring' := 'call'}
PROPERTY Error : BOOL
GET
Error := _Error;
END_GET
END_PROPERTY

{attribute 'monitoring' := 'call'}
PROPERTY ErrorId : UDINT
GET
ErrorID := _ErrorID;
END_GET
END_PROPERTY

METHOD Reset
VAR_INPUT
	Module : I_Module;
END_VAR
_Error	 := FALSE;
_ErrorId := 0;
_Busy	 := FALSE;
Module.Accept(THIS^);
IF __QUERYINTERFACE(Module, Resettable) THEN
	Resettable.Reset();
END_IF

IF __QUERYINTERFACE(Module, Result) THEN
	IF Result.Error THEN
		_Error	 := TRUE;
		_ErrorId := Result.ErrorId;
	END_IF

	IF Result.Busy THEN
		_Busy := TRUE;
	END_IF
END_IF
END_METHOD

METHOD VisitComponent
VAR_INPUT
	Component : I_Component;
END_VAR
IF __QUERYINTERFACE(Component, Resettable) THEN
	Resettable.Reset();
END_IF

IF __QUERYINTERFACE(Component, Result) THEN
	IF Result.Error THEN
		ErrorComponent := Component;
		_Error		   := TRUE;
		_ErrorId	   := Result.ErrorId;
	END_IF

	IF Result.Busy THEN
		_Busy := TRUE;
	END_IF
END_IF
END_METHOD

METHOD VisitModule
VAR_INPUT
	Module : I_Module;
END_VAR
Module.Components.Accept(THIS^);
Module.Modules.Accept(THIS^);
IF __QUERYINTERFACE(Module, Resettable) THEN
	Resettable.Reset();
END_IF

IF __QUERYINTERFACE(Module, Result) THEN
	IF Result.Error THEN
		ErrorModule := Module;
		_Error		:= TRUE;
		_ErrorId	:= Result.ErrorId;
	END_IF

	IF Result.Busy THEN
		_Busy := TRUE;
	END_IF
END_IF
END_METHOD

END_FUNCTION_BLOCK

// ---- Visitors/Statemachine/ChangeModeOnAllSubModulesVisitor.TcPOU
FUNCTION_BLOCK ChangeModeOnAllSubModulesVisitor IMPLEMENTS I_ModuleVisitor
VAR
	TargetMode	 : DINT;
	Statemachine : I_ContainStatemachine;
END_VAR

METHOD ChangeMode
VAR_INPUT
	TargetMode : DINT;
	Module	   : I_Module;
END_VAR
THIS^.TargetMode := TargetMode;
Module.Modules.Accept(THIS^);
END_METHOD

METHOD VisitModule
VAR_INPUT
	Module : I_Module;
END_VAR
IF __QUERYINTERFACE(Module, Statemachine) THEN
	Statemachine.Statemachine.Mode.ChangeMode(THIS^.TargetMode);
END_IF
END_METHOD

END_FUNCTION_BLOCK

// ---- Visitors/Statemachine/ChangeStateOnAllSubModulesVisitor.TcPOU
FUNCTION_BLOCK ChangeStateOnAllSubModulesVisitor IMPLEMENTS I_ModuleVisitor
VAR
	TargetState	 : DINT;
	Statemachine : I_ContainStatemachine;
	StateChanged : BOOL;
END_VAR

METHOD ChangeState : BOOL
VAR_INPUT
	TargetState : DINT;
	Module		: I_Module;
END_VAR
StateChanged	  := TRUE;
THIS^.TargetState := TargetState;
Module.Modules.Accept(THIS^);
ChangeState := StateChanged;
END_METHOD

METHOD VisitModule
VAR_INPUT
	Module : I_Module;
END_VAR

VAR_INST
	ReturnModule : I_Module;
END_VAR
IF __QUERYINTERFACE(Module, Statemachine) THEN
	IF Statemachine.Statemachine = 0 THEN
		ReturnModule := Module;
		RETURN;
	END_IF

	Statemachine.Statemachine.ChangeState(THIS^.TargetState);
	IF Statemachine.Statemachine.CurrentState <> THIS^.TargetState THEN
		StateChanged := FALSE;
	END_IF
END_IF
END_METHOD

END_FUNCTION_BLOCK

// ---- Visitors/Statemachine/EventReactorVisitor.TcPOU
FUNCTION_BLOCK EventReactorVisitor EXTENDS CyclicComponent IMPLEMENTS I_ModuleVisitor, I_ComponentVisitor
VAR
	EntryModule			 : I_Module;
	HighestEventReaction : DINT;
	EventReaction		 : I_EventReaction;
	ModuleStatemachine	 : I_ContainStatemachine;
END_VAR

METHOD CyclicLogic
IF ModuleStatemachine = 0 THEN
	RETURN;
END_IF

HighestEventReaction := 0;
EntryModule.Accept(THIS^);
CASE HighestEventReaction OF
	0: // Verbose
	1: // Info
	2: // Warning
	3: // Error
	4: // Critical
END_CASE
END_METHOD

(*FB_Init is always available implicitly and it is used primarily for initialization.
The return value is not evaluated. For a specific influence, you can also declare the
methods explicitly and provide additional code there with the standard initialization
code. You can evaluate the return value.*)
METHOD FB_Init : BOOL
VAR_INPUT
	(* TRUE: the retain variables are initialized (reset warm / reset cold)*)
	bInitRetains : BOOL;

	(* TRUE: the instance will be copied to the copy code afterward (online change)   *)
	bInCopyCode : BOOL;
	Name		: T_MaxString;
	EntryModule : I_Module;
END_VAR
THIS^.EntryModule := EntryModule;
__QUERYINTERFACE(EntryModule, ModuleStatemachine);
END_METHOD

METHOD VisitComponent
VAR_INPUT
	Component : I_Component;
END_VAR

VAR
	Reaction : DINT;
END_VAR
IF __QUERYINTERFACE(Component, EventReaction) THEN
	Reaction := EventReaction.GetHighestActiveEventReaction();
	IF Reaction > HighestEventReaction THEN
		HighestEventReaction := Reaction;
	END_IF
END_IF
END_METHOD

METHOD VisitModule
VAR_INPUT
	Module : I_Module;
END_VAR

VAR
	Reaction : DINT;
END_VAR
Module.Components.Accept(THIS^);
Module.Modules.Accept(THIS^);
IF __QUERYINTERFACE(Module, EventReaction) THEN
	Reaction := EventReaction.GetHighestActiveEventReaction();
	IF Reaction > HighestEventReaction THEN
		HighestEventReaction := Reaction;
	END_IF
END_IF
END_METHOD

END_FUNCTION_BLOCK

// ---- Visitors/Stop/StopAllComponentsVisitor.TcPOU
FUNCTION_BLOCK StopAllComponentsVisitor IMPLEMENTS I_ComponentVisitor
VAR
	Stoppable : I_Stoppable;
	_Stopped  : BOOL;
END_VAR

METHOD Stop
VAR_INPUT
	Components : I_ComponentCollection;
END_VAR
_Stopped := TRUE;
Components.Accept(THIS^);
END_METHOD

{attribute 'monitoring' := 'call'}
PROPERTY Stopped : BOOL
GET
Stopped := _Stopped;
END_GET
END_PROPERTY

METHOD VisitComponent
VAR_INPUT
	Component : I_Component;
END_VAR
IF __QUERYINTERFACE(Component, Stoppable) THEN
	IF NOT Stoppable.Stopped THEN
		Stoppable.Stop();
		_Stopped := FALSE;
	END_IF
END_IF
END_METHOD

END_FUNCTION_BLOCK

// ---- _Internal/CollectionPeeker/CollectionPeeker.TcPOU
{attribute 'hide_all_locals'}
FUNCTION_BLOCK CollectionPeeker
VAR_GENERIC CONSTANT
	Peek_Size : UDINT := 5;
END_VAR IMPLEMENTS I_CollectionPeeker, I_Peeker
VAR
	_CurrentItem	: UDINT;
	_EndItem		: UDINT;
	_CollectionName : T_MaxString;
	_Collection		: I_Collection;
	_Items			: ARRAY[1..Peek_Size] OF I_Base;
END_VAR

{attribute 'monitoring':='call'}
PROPERTY CollectionName : T_MaxString
GET
CollectionName := _CollectionName;
END_GET
SET
_CollectionName := CollectionName;
END_SET
END_PROPERTY

{attribute 'monitoring' := 'call'}
PROPERTY FirstItem : UDINT
GET
FirstItem := _CurrentItem;
END_GET
SET
IF _Collection = 0 THEN
	RETURN;
END_IF

IF FirstItem > _Collection.Count OR FirstItem < 1 THEN
	RETURN;
END_IF

_CurrentItem := FirstItem;
UpdateEndItem();
RefreshItems();
END_SET
END_PROPERTY

{attribute 'monitoring' := 'call'}
PROPERTY Items : REFERENCE TO ARRAY[1..Peek_Size] OF I_Base
GET
Items REF= _Items;
END_GET
END_PROPERTY

{attribute 'monitoring' := 'call'}
PROPERTY LastItem : UDINT
GET
LastItem := _EndItem;
END_GET
END_PROPERTY

{attribute 'monitoring' := 'call'}
PROPERTY MoveDownOne : BOOL
GET
END_GET
SET
IF _Collection = 0 OR NOT MoveDownOne THEN
	RETURN;
END_IF

IF _Collection.Count <= Peek_Size THEN
	RETURN;
END_IF

_CurrentItem := _CurrentItem + 1;
IF _CurrentItem > _Collection.Count THEN
	_CurrentItem := 1;
END_IF

UpdateEndItem();
RefreshItems();
END_SET
END_PROPERTY

{attribute 'monitoring' := 'call'}
PROPERTY MoveUpOne : BOOL
GET
END_GET
SET
IF _Collection = 0 THEN
	RETURN;
END_IF

IF _Collection.Count <= Peek_Size THEN
	RETURN;
END_IF

_CurrentItem := _CurrentItem - 1;
IF _CurrentItem < 1 THEN
	_CurrentItem := _Collection.Count;
END_IF

UpdateEndItem();
RefreshItems();
END_SET
END_PROPERTY

{attribute 'monitoring' := 'call'}
PROPERTY PageDown : BOOL
GET
END_GET
SET
IF _Collection = 0 OR NOT PageDown THEN
	RETURN;
END_IF

IF _Collection.Count <= Peek_Size THEN
	RETURN;
END_IF

IF _CurrentItem > (_Collection.Count - Peek_Size) THEN
	_CurrentItem := (Peek_Size - (_Collection.Count - _CurrentItem));
ELSE
	_CurrentItem := _CurrentItem + Peek_Size;
END_IF

UpdateEndItem();
RefreshItems();
END_SET
END_PROPERTY

{attribute 'monitoring' := 'call'}
PROPERTY PageUp : BOOL
GET
END_GET
SET
VAR
	tmp : UDINT;
END_VAR
IF _Collection = 0 OR NOT PageUp THEN
	RETURN;
END_IF

IF _Collection.Count <= Peek_Size THEN
	RETURN;
END_IF

IF _CurrentItem < Peek_Size THEN
	_CurrentItem := (_Collection.Count - (Peek_Size - _CurrentItem));
ELSE
	_CurrentItem := _CurrentItem - Peek_Size;
END_IF

UpdateEndItem();
RefreshItems();
END_SET
END_PROPERTY

METHOD PeekAt
VAR_INPUT
	Peekable : I_Peekable;
END_VAR
Peekable.AcceptPeeker(THIS^);
END_METHOD

METHOD PeekCollection
VAR_INPUT
	Collection : I_Collection;
END_VAR
_Collection	 := Collection;
_CurrentItem := 1;
_EndItem	 := Peek_Size;
RefreshItems();
END_METHOD

{attribute 'monitoring':='call'}
PROPERTY Refresh : BOOL
GET
END_GET
SET
IF _Collection <> 0 AND Refresh THEN
	RefreshItems();
END_IF
END_SET
END_PROPERTY

METHOD PRIVATE RefreshItems
VAR
	startItem  : UDINT;
	endItem	   : UDINT;
	i		   : UDINT := 1;
	wrapAround : BOOL;
END_VAR
MEMSET(ADR(_Items), 0, SIZEOF(_Items));
IF _CurrentItem > _EndItem THEN //we're wrapped around
	i		   := 1 + ((_Collection.Count - _CurrentItem) + 1);
	wrapAround := TRUE;
END_IF

_Collection.ResetIterator();
WHILE _Collection.MoveToNext DO
	IF _Collection.CurrentItem >= _CurrentItem AND _Collection.CurrentItem <= _EndItem THEN
		_Items[i] := _Collection.Current;
		i		  := i + 1;
	ELSIF wrapAround AND (_Collection.CurrentItem >= _CurrentItem OR _Collection.CurrentItem <= _EndItem) THEN
		_Items[i] := _Collection.Current;
		i		  := i + 1;
		IF i > Peek_Size THEN
			i := 1;
		END_IF
	END_IF
END_WHILE
END_METHOD

METHOD PRIVATE UpdateEndItem
VAR_INPUT
END_VAR
_EndItem := _CurrentItem + Peek_Size - 1;
IF _EndItem > _Collection.Count THEN
	_EndItem := _EndItem - _Collection.Count;
END_IF
END_METHOD

METHOD PRIVATE UpdateFirstItem
VAR_INPUT
END_VAR
END_METHOD

END_FUNCTION_BLOCK

// ---- _Internal/List/List.TcPOU
FUNCTION_BLOCK List
VAR_GENERIC CONSTANT
	ListSize : UDINT := 2;
END_VAR
EXTENDS Collection<ListSize> IMPLEMENTS I_List
VAR
	_ListCount : UDINT := 0;
END_VAR

METHOD AddItem
VAR_INPUT
	Item : I_Base;
END_VAR
SUPER^.AddItem(Item);
CountListItems();
END_METHOD

METHOD Clear
SUPER^.Clear();
CountListItems();
END_METHOD

METHOD ContainsItem : BOOL
VAR_INPUT
	Item : I_Base;
END_VAR

VAR
	i	  : UDINT;
	pItem : POINTER TO I_Base;
END_VAR
IF Item = 0 THEN
	Trace.LogMessage(InstancePath, 'Item is not a valid interface!');
	RETURN;
END_IF

IF _ListCount = 0 THEN
	RETURN;
END_IF

FOR i := 0 TO (_ListCount - 1) DO
	IF _Data[i] = Item AND _Data[i] <> 0 THEN
		ContainsItem := TRUE;
		RETURN;
	END_IF
END_FOR
END_METHOD

{attribute 'monitoring' := 'call'}
PROPERTY Count : UDINT
GET
Count := _ListCount;
END_GET
END_PROPERTY

METHOD PRIVATE CountListItems
VAR
	i	  : UDINT;
	pItem : POINTER TO I_Base;
END_VAR
IF _Count = 0 THEN
	_ListCount := 0;
	RETURN;
END_IF

_ListCount := 0;
FOR i := 0 TO (_Count - 1) DO
	IF _Data[i] <> 0 THEN
		_ListCount := _ListCount + 1;
	END_IF
END_FOR
END_METHOD

METHOD GetAtIndex : I_Base
VAR_INPUT
	Index : UDINT;
END_VAR

VAR
	pItem : POINTER TO I_Base;
END_VAR
IF Count = 0 THEN
	Trace.LogMessage(InstancePath, 'No Items found in this List!');
	RETURN;
END_IF

IF Index > (_Count - 1) THEN
	Trace.LogMessage(InstancePath, 'Index does not exist in List!');
	RETURN;
END_IF

GetAtIndex := _Data[Index];
END_METHOD

METHOD InsertAtIndex : BOOL
VAR_INPUT
	Item  : I_Base;
	Index : UDINT;
END_VAR

VAR
	pItem	  : POINTER TO I_Base;
	pItemNext : POINTER TO I_Base;
	i		  : UDINT;
END_VAR
IF Index > _Count THEN
	InsertAtIndex := FALSE;
	RETURN;
END_IF

_Count := (_Count + 1);
FOR i := _Count TO Index + 1 BY -1 DO
	_Data[i] := _Data[i - 1];
END_FOR

_Data[Index] := Item;
CountListItems();
END_METHOD

METHOD RemoveAtIndex
VAR_INPUT
	Index : UDINT;
END_VAR

VAR
	pItem : POINTER TO I_Base;
END_VAR
IF Count = 0 THEN
	Trace.LogMessage(InstancePath, 'No Items found in this List!');
	RETURN;
END_IF

IF Index > (_Count - 1) THEN
	Trace.LogMessage(InstancePath, 'Index does not exist in List!');
	RETURN;
END_IF

MEMMOVE(ADR(_Data[Index]), ADR(_Data[Index + 1]), (_Count - Index - 1) * SIZEOF(PVOID));
_Count := _Count - 1;

//pItem  := Collection.pBuffer + (Index * SIZEOF(PVOID));
CountListItems();
END_METHOD

METHOD RemoveItem
VAR_INPUT
	Item : I_Base;
END_VAR

VAR
	pItem		 : POINTER TO I_Base;
	pItemNext	 : POINTER TO I_Base;
	i			 : UDINT;
	removedItems : UDINT;
END_VAR
IF _Count = 0 THEN
	Trace.LogMessage(InstancePath, 'No Items found in this Collection!');
	RETURN;
END_IF

IF Item = 0 THEN
	Trace.LogMessage(InstancePath, 'Item to remove needs to be valid interface!');
	RETURN;
END_IF

